    G_SystemInfo.DeviceName := SystemParameters.o_DeviceName;
    G_SystemInfo.HWVersion := SystemParameters.o_HardwareVersion;
    G_SystemInfo.SWVersion := SystemParameters.o_SoftwareVersion;
    G_SystemInfo.Identity.ProductCode := SystemParameters.o_ProductCode;    (* Type for control unit. *)
    G_SystemInfo.Identity.Revision := SystemParameters.o_RevisionNumber;      (* Revision for control unit *)
    G_SystemInfo.Identity.SerialNumber := SystemParameters.o_SerialNumber;  (* Serial number for control unit *)
    G_SystemInfo.Identity.VendorId := SystemParameters.o_VendorId;               (* Vendor id which is read from firmware *)
          
    G_SystemInfo.MACAddress := SystemParameters.o_MAC;
    G_SystemInfo.EthernetConfiguration :=  SystemParameters.i_Ethernet;
    G_SystemInfo.CAN1_Comms := SystemParameters.i_CAN1;
    G_SystemInfo.CAN2_Comms := SystemParameters.i_CAN2;
    G_SystemInfo.CAN3_Comms := SystemParameters.i_CAN3;
    G_SystemInfo.CAN4_Comms := SystemParameters.i_CAN4;
    
    (* Get 5050 fw error log pointer *)
    SystemErrorLog.init();
    G_SystemInfo.FWErrorLog :=  SystemErrorLog.o_ErrorLog;


    
END_IF
END_ACTION

ACTION Init_Events_Action:
(*###########################################################*)
(*This block is created implicit. Don't add own code to here.*)
(*###########################################################*)
;



G_InitEventsReady:=TRUE;
END_ACTION

ACTION Init_Exit_Action:
(*###########################################################*)
(*This block is created implicit. Don't add own code to here.*)
(*###########################################################*)
;


G_InitExitReady:=TRUE;
END_ACTION

ACTION Init_Flash_Action:
(*###########################################################*)
(*This block is created implicit. Don't add own code to here.*)
(*###########################################################*)

  	(* Get info for MRAM area used for programmer. *)
  	SYSTEM_SHM_MRAM_GET_IEC_AREA(ADR(G_ShmUserMRAM));
  	(* Check addresses and divide area between parameter system and are available for user *)
	IF ((G_ShmUserMRAM.endAddress > 0) AND (G_ShmUserMRAM.startAddress > 0))
		AND (G_ShmUserMRAM.endAddress > (G_ShmUserMRAM.startAddress + G_MRAM_AREA_SIZE_FOR_PAR_SYS + 100)) THEN
		(* Init file system for parameters *)
		(* Init ParameterHandler to use MRAM *)
        G_Common.ParHandler.Init(i_pParamArea:=G_ShmUserMRAM.startAddress,
            i_ParamAreaSize:=G_MRAM_AREA_SIZE_FOR_PAR_SYS ,
            i_Keyword:=G_PARAMHANDLERKEYWORD ,
            i_ParameterMaxDataSize:= G_PARAM_BLOCK_MAX_SIZE);
		(* Set user MRAM pointers, which tells area for freely used by programmer. *)
		G_MramStartAddressForUser := G_ShmUserMRAM.startAddress + G_MRAM_AREA_SIZE_FOR_PAR_SYS;
		G_MramEndAddressForUser := G_ShmUserMRAM.endAddress ;
	ELSE
		(* Error *)
		G_MramInitErrors := - 1;
	END_IF
	
	(* Init user MRAM structure*)
	IF (0 <> G_ShmUserMRAM.startAddress) AND (G_ShmUserMRAM.reservedSize >= (SIZEOF(UserMramStructure) + DWORD_TO_DINT(G_MRAM_AREA_SIZE_FOR_PAR_SYS))) THEN
		G_pUserMramStructure := G_MramStartAddressForUser;
		IF G_pUserMramStructure^.UserMRAMTag = 16#AA55AA55 THEN
			G_pUserMramStructure^.UserMRAMdataValid := TRUE;
			G_pUserMramStructure^.UserMRAMinitError := 0;
		ELSE
			G_pUserMramStructure^.UserMRAMdataValid := FALSE;
			G_pUserMramStructure^.UserMRAMTag := 16#AA55AA55;
			G_pUserMramStructure^.UserMRAMinitError := 2; 
		END_IF 
	END_IF
	
	
G_InitFlashReady:=TRUE;
END_ACTION

ACTION Init_IO_Action:
(*###########################################################*)
(*This block is created implicit. Don't add own code to here.*)
(*###########################################################*)
;
(*IO init:*)
(*IO_Init functions*)
		(* Force ref always ON *)
		REF_OUT_5V_Enable:=TRUE;
		REF_OUT_10V_Enable:=TRUE;

(*#########################################*)
(* INIT FOR AI Channel 1 X1.09*)

AI_SET_PU_u16_DrivetrainTemp_AI := FALSE;


    AI_SET_mA_u16_DrivetrainTemp_AI := FALSE;

    G_AIprotection_X1_09(i_Enable := TRUE, i_AiInmAMode:= FALSE);


(*#########################################*)
(* INIT FOR AI Channel 20 X1.10*)

    AI_SET_PU_u16_ChargePlugPresent_AI := FALSE;


    AI_SET_mA_u16_ChargePlugPresent_AI := FALSE;

    G_AIprotection_X1_10(i_Enable := TRUE, i_AiInmAMode:= FALSE);


(*##################################################################################*)
(* INIT FOR PULSE INPUT CHANNEL 22 Pin 1.11*)

PI_INIT_ERROR_q_BatteryInterlockIn_DI := IO_PULSEIN_SET_CONFIG(
	i_Mode:=IO_PULSEIN_MODE_DI,
	i_ChannelNbr:=22,
	i_ResetChnNbr:=0,
	i_ChannelPairNbr:=0,
	i_EdgeSelect:=0,
	i_EdgePolarity:=0,
	i_Filter:=0,
	i_GateTime:=100);
   IF NOT ( PI_INIT_ERROR_q_BatteryInterlockIn_DI = 0 ) THEN
         ERR_FLAG_IO_INIT := TRUE;
    END_IF

(*#########################################*)
(* INIT FOR PWFM CHANNEL 9 Pin 1.12*)

    PWFM_ERROR_INIT_q_BackupPump_DO :=  IO_PWFM_SET_CONFIG(
		i_PwfmMode:=IO_PWFM_MODE_DIGITAL_OUTPUT,
		i_PwfmChn:=9,
		i_OverCurrentLimit := 1000,
		i_SupplyVoltage:=0,
		i_CoilResistance:=0,
		i_CorrectionGain:=0,
		i_DiagnosticTimeDelay:=0);
   IF NOT ( PWFM_ERROR_INIT_q_BackupPump_DO = 0 ) THEN
         ERR_FLAG_IO_INIT := TRUE;
    END_IF
    DO_q_BackupPump_DO := FALSE;

(*#########################################*)
(* INIT FOR AI Channel 2 X1.20*)

    AI_SET_PU_u16_Heater1Temperature_AI := FALSE;


    AI_SET_mA_u16_Heater1Temperature_AI := FALSE;

    G_AIprotection_X1_20(i_Enable := TRUE, i_AiInmAMode:= FALSE);


(*#########################################*)
(* INIT FOR AI Channel 21 X1.21*)

    AI_SET_PU_u16_Heater2Temperature_AI := FALSE;


    AI_SET_mA_u16_Heater2Temperature_AI := FALSE;

    G_AIprotection_X1_21(i_Enable := TRUE, i_AiInmAMode:= FALSE);


(*#########################################*)
(* INIT FOR PWFM CHANNEL 21 Pin 1.22*)

    PWFM_ERROR_INIT_q_BatteryDischargeMain_DO := IO_PWFM_SET_CONFIG(
	i_PwfmMode:=IO_PWFM_MODE_DIGITAL_OUTPUT,
	i_PwfmChn:=21,
	i_OverCurrentLimit := 0,
	i_SupplyVoltage:=0,
	i_CoilResistance:=0,
	i_CorrectionGain:=0,
	i_DiagnosticTimeDelay:=0);
   IF NOT ( PWFM_ERROR_INIT_q_BatteryDischargeMain_DO = 0 ) THEN
         ERR_FLAG_IO_INIT := TRUE;
    END_IF
    DO_q_BatteryDischargeMain_DO := FALSE;

(*#########################################*)
(* INIT FOR PWFM CHANNEL 10 Pin 1.23*)

    PWFM_ERROR_INIT_q_AirPressureReliefValve_DO := IO_PWFM_SET_CONFIG(
	i_PwfmMode:=IO_PWFM_MODE_DIGITAL_OUTPUT,
	i_PwfmChn:=10,
	i_OverCurrentLimit := 1000,
	i_SupplyVoltage:=0,
	i_CoilResistance:=0,
	i_CorrectionGain:=0,
	i_DiagnosticTimeDelay:=0);
   IF NOT ( PWFM_ERROR_INIT_q_AirPressureReliefValve_DO = 0 ) THEN
         ERR_FLAG_IO_INIT := TRUE;
    END_IF
    DO_q_AirPressureReliefValve_DO := FALSE;

(*#########################################*)
(* INIT FOR PWFM CHANNEL 28 Pin 1.29*)

    PWFM_ERROR_INIT_q_Battery1ChargePrecharge_DO:= IO_PWFM_SET_CONFIG(
	i_PwfmMode:=IO_PWFM_MODE_DIGITAL_OUTPUT,
	i_PwfmChn:=28,
	i_OverCurrentLimit := 0,
	i_SupplyVoltage:=0,
	i_CoilResistance:=0,
	i_CorrectionGain:=0,
	i_DiagnosticTimeDelay:=0);
   IF NOT ( PWFM_ERROR_INIT_q_Battery1ChargePrecharge_DO = 0 ) THEN
         ERR_FLAG_IO_INIT := TRUE;
    END_IF
    DO_q_Battery1ChargePrecharge_DO := FALSE;

(*#########################################*)
(* INIT FOR PWFM CHANNEL 27 Pin 1.30*)

    PWFM_ERROR_INIT_q_Battery1ChargeMain_DO:= IO_PWFM_SET_CONFIG(
	i_PwfmMode:=IO_PWFM_MODE_DIGITAL_OUTPUT,
	i_PwfmChn:=27,
	i_OverCurrentLimit := 0,
	i_SupplyVoltage:=0,
	i_CoilResistance:=0,
	i_CorrectionGain:=0,
	i_DiagnosticTimeDelay:=0);
   IF NOT ( PWFM_ERROR_INIT_q_Battery1ChargeMain_DO = 0 ) THEN
         ERR_FLAG_IO_INIT := TRUE;
    END_IF
    DO_q_Battery1ChargeMain_DO := FALSE;

(*#########################################*)
(* INIT FOR PWFM CHANNEL 26 Pin 1.31*)

    PWFM_ERROR_INIT_q_Battery2ChargePrecharge_DO := IO_PWFM_SET_CONFIG(
	i_PwfmMode:=IO_PWFM_MODE_DIGITAL_OUTPUT,
	i_PwfmChn:=26,
	i_OverCurrentLimit := 0,
	i_SupplyVoltage:=0,
	i_CoilResistance:=0,
	i_CorrectionGain:=0,
	i_DiagnosticTimeDelay:=0);
   IF NOT ( PWFM_ERROR_INIT_q_Battery2ChargePrecharge_DO = 0 ) THEN
         ERR_FLAG_IO_INIT := TRUE;
    END_IF
    DO_q_Battery2ChargePrecharge_DO := FALSE;

(*#########################################*)
(* INIT FOR PWFM CHANNEL 25 Pin 1.32*)

    PWFM_ERROR_INIT_q_DrivetrainInverterTorqueless_DO := IO_PWFM_SET_CONFIG(
	i_PwfmMode:=IO_PWFM_MODE_DIGITAL_OUTPUT,
	i_PwfmChn:=25,
	i_OverCurrentLimit := 0,
	i_SupplyVoltage:=0,
	i_CoilResistance:=0,
	i_CorrectionGain:=0,
	i_DiagnosticTimeDelay:=0);
   IF NOT ( PWFM_ERROR_INIT_q_DrivetrainInverterTorqueless_DO = 0 ) THEN
         ERR_FLAG_IO_INIT := TRUE;
    END_IF
    DO_q_DrivetrainInverterTorqueless_DO := FALSE;

(*#########################################*)
(* INIT FOR PWFM CHANNEL 23 Pin 1.33*)

    PWFM_ERROR_INIT_q_BatteryDischargePrecharge_DO := IO_PWFM_SET_CONFIG(
	i_PwfmMode:=IO_PWFM_MODE_DIGITAL_OUTPUT,
	i_PwfmChn:=23,
	i_OverCurrentLimit := 0,
	i_SupplyVoltage:=0,
	i_CoilResistance:=0,
	i_CorrectionGain:=0,
	i_DiagnosticTimeDelay:=0);

   IF NOT ( PWFM_ERROR_INIT_q_BatteryDischargePrecharge_DO = 0 ) THEN
         ERR_FLAG_IO_INIT := TRUE;
    END_IF
	DO_q_BatteryDischargePrecharge_DO := FALSE;

(*#########################################*)
(* INIT FOR PWFM CHANNEL 24 Pin 1.34*)

    PWFM_ERROR_INIT_u32_DynamoFrequency_PWFM := IO_PWFM_SET_CONFIG(
	i_PwfmMode:=IO_PWFM_MODE_DIRECT_PWFM,
	i_PwfmChn:=24,
	i_OverCurrentLimit :=0,
	i_SupplyVoltage:=0,
	i_CoilResistance:=0,
	i_CorrectionGain:=0,
	i_DiagnosticTimeDelay:=0);
   IF NOT ( PWFM_ERROR_INIT_u32_DynamoFrequency_PWFM = 0 ) THEN
         ERR_FLAG_IO_INIT := TRUE;
    END_IF
    PWFM_FREQ_u32_DynamoFrequency_PWFM :=     200;
    PWFM_RATIO_u32_DynamoFrequency_PWFM := 0;

(*#########################################*)
(* INIT FOR PWFM CHANNEL 22 Pin 1.35*)

    PWFM_ERROR_INIT_q_Battery2ChargeMain_DO := IO_PWFM_SET_CONFIG(
	i_PwfmMode:=IO_PWFM_MODE_DIGITAL_OUTPUT,
	i_PwfmChn:=22,
	i_OverCurrentLimit := 0,
	i_SupplyVoltage:=0,
	i_CoilResistance:=0,
	i_CorrectionGain:=0,
	i_DiagnosticTimeDelay:=0);
   IF NOT ( PWFM_ERROR_INIT_q_Battery2ChargeMain_DO = 0 ) THEN
         ERR_FLAG_IO_INIT := TRUE;
    END_IF
    DO_q_Battery2ChargeMain_DO := FALSE;

(*##################################################################################*)
(* INIT FOR PULSE INPUT CHANNEL 1 Pin 2.6*)

PI_INIT_ERROR_q_Battery1ChargeRq_DI := IO_PULSEIN_SET_CONFIG(
	i_Mode:=IO_PULSEIN_MODE_1CH,
	i_ChannelNbr:=1,
	i_ResetChnNbr:=0,
	i_ChannelPairNbr:=0,
	i_EdgeSelect:=0,
	i_EdgePolarity:=0,
	i_Filter:=0,
	i_GateTime:=100);
   IF NOT ( PI_INIT_ERROR_q_Battery1ChargeRq_DI = 0 ) THEN
         ERR_FLAG_IO_INIT := TRUE;
    END_IF

(*##################################################################################*)
(* INIT FOR PULSE INPUT CHANNEL 2 Pin 2.7*)

    PI_INIT_ERROR_q_Battery1DiscahrgeRq_DI := IO_PULSEIN_SET_CONFIG(
	i_Mode:=IO_PULSEIN_MODE_1CH,
	i_ChannelNbr:=2,
	i_ResetChnNbr:=0,
	i_ChannelPairNbr:=0,
	i_EdgeSelect:=0,
	i_EdgePolarity:=0,
	i_Filter:=0,
	i_GateTime:=100);
    IF NOT ( PI_INIT_ERROR_q_Battery1DiscahrgeRq_DI = 0 ) THEN
         ERR_FLAG_IO_INIT := TRUE;
    END_IF

(*##################################################################################*)
(* INIT FOR PULSE INPUT CHANNEL 3 Pin 2.8*)

    PI_INIT_ERROR_q_Battery2ChargeRq_DI := IO_PULSEIN_SET_CONFIG(
	i_Mode:=IO_PULSEIN_MODE_1CH,
	i_ChannelNbr:=3,
	i_ResetChnNbr:=0,
	i_ChannelPairNbr:=0,
	i_EdgeSelect:=0,
	i_EdgePolarity:=0,
	i_Filter:=0,
	i_GateTime:=100);
   IF NOT ( PI_INIT_ERROR_q_Battery2ChargeRq_DI = 0 ) THEN
         ERR_FLAG_IO_INIT := TRUE;
    END_IF

(*##################################################################################*)
(* INIT FOR PULSE INPUT CHANNEL 4 Pin 2.9*)

    PI_INIT_ERROR_q_Batter2DischargeRq_DI := IO_PULSEIN_SET_CONFIG(
	i_Mode:=IO_PULSEIN_MODE_1CH,
	i_ChannelNbr:=4,
	i_ResetChnNbr:=0,
	i_ChannelPairNbr:=0,
	i_EdgeSelect:=0,
	i_EdgePolarity:=0,
	i_Filter:=0,
	i_GateTime:=100);
   IF NOT ( PI_INIT_ERROR_q_Batter2DischargeRq_DI = 0 ) THEN
         ERR_FLAG_IO_INIT := TRUE;
    END_IF

(*#########################################*)
(* INIT FOR PWFM CHANNEL 12 Pin 2.13*)

    PWFM_ERROR_INIT_q_ChargePlugLockPulse_DO := IO_PWFM_SET_CONFIG(
	i_PwfmMode:=IO_PWFM_MODE_DIGITAL_OUTPUT,
	i_PwfmChn:=12,
	i_OverCurrentLimit := 1000,
	i_SupplyVoltage:=0,
	i_CoilResistance:=0,
	i_CorrectionGain:=0,
	i_DiagnosticTimeDelay:=0);
    IF NOT ( PWFM_ERROR_INIT_q_ChargePlugLockPulse_DO = 0 ) THEN
         ERR_FLAG_IO_INIT := TRUE;
    END_IF
    DO_q_ChargePlugLockPulse_DO := FALSE;

(*#########################################*)
(* INIT FOR PWFM CHANNEL 11 Pin 2.14*)

    PWFM_ERROR_INIT_q_ChargePlugLockPosition_DO := IO_PWFM_SET_CONFIG(
	i_PwfmMode:=IO_PWFM_MODE_DIGITAL_OUTPUT,
	i_PwfmChn:=11,
	i_OverCurrentLimit := 1000,
	i_SupplyVoltage:=0,
	i_CoilResistance:=0,
	i_CorrectionGain:=0,
	i_DiagnosticTimeDelay:=0);
    IF NOT ( PWFM_ERROR_INIT_q_ChargePlugLockPosition_DO = 0 ) THEN
         ERR_FLAG_IO_INIT := TRUE;
    END_IF
    DO_q_ChargePlugLockPosition_DO := FALSE;

(*##################################################################################*)
(* INIT FOR PULSE INPUT CHANNEL 5 Pin 2.15*)

(*##################################################################################*)
(* INIT FOR PULSE INPUT CHANNEL 9 Pin 2.16*)

    PI_ERROR_q_ChargePlugLockStatus_DI := IO_PULSEIN_SET_CONFIG(
	i_Mode:=IO_PULSEIN_MODE_1CH,
	i_ChannelNbr:=9,
	i_ResetChnNbr:=0,
	i_ChannelPairNbr:=0,
	i_EdgeSelect:=0,
	i_EdgePolarity:=0,
	i_Filter:=0,
	i_GateTime:=100);
   IF NOT ( PI_ERROR_q_ChargePlugLockStatus_DI = 0 ) THEN
         ERR_FLAG_IO_INIT := TRUE;
    END_IF


(*##################################################################################*)
(* INIT FOR PULSE INPUT CHANNEL 10 Pin 2.17*)

(*##################################################################################*)
(* INIT FOR PULSE INPUT CHANNEL 6 Pin 2.18*)

(*##################################################################################*)
(* INIT FOR PULSE INPUT CHANNEL 11 Pin 2.19*)

(*##################################################################################*)
(* INIT FOR PULSE INPUT CHANNEL 12 Pin 2.20*)

(*#########################################*)
(* INIT FOR AI Channel 3 X2.23*)

    AI_SET_PU_u16_HeaterDiagnose_AI := FALSE;


    AI_SET_mA_u16_HeaterDiagnose_AI := FALSE;

    G_AIprotection_X2_23(i_Enable := TRUE, i_AiInmAMode:= FALSE);


(*#########################################*)
(* INIT FOR  SINKING DIGITAL OUTPUT 2.26*)

(*#########################################*)
(* INIT FOR  SINKING DIGITAL OUTPUT 2.27*)

(*#########################################*)
(* INIT FOR PWFM CHANNEL 14 Pin 2.28*)

    PWFM_ERROR_INIT_q_DrivetrainKL15D_DO := IO_PWFM_SET_CONFIG(
	i_PwfmMode:=IO_PWFM_MODE_DIGITAL_OUTPUT,
	i_PwfmChn:=14,
	i_OverCurrentLimit := 1000,
	i_SupplyVoltage:=0,
	i_CoilResistance:=0,
	i_CorrectionGain:=0,
	i_DiagnosticTimeDelay:=0);
    IF NOT ( PWFM_ERROR_INIT_q_DrivetrainKL15D_DO = 0 ) THEN
         ERR_FLAG_IO_INIT := TRUE;
    END_IF
    DO_q_DrivetrainKL15D_DO := FALSE;

(*#########################################*)
(* INIT FOR PWFM CHANNEL 13 Pin 2.29*)

    PWFM_ERROR_INIT_q_DrivetrainKL15C_DO := IO_PWFM_SET_CONFIG(
	i_PwfmMode:=IO_PWFM_MODE_DIGITAL_OUTPUT,
	i_PwfmChn:=13,
	i_OverCurrentLimit := 1000,
	i_SupplyVoltage:=0,
	i_CoilResistance:=0,
	i_CorrectionGain:=0,
	i_DiagnosticTimeDelay:=0);
    IF NOT ( PWFM_ERROR_INIT_q_DrivetrainKL15C_DO = 0 ) THEN
         ERR_FLAG_IO_INIT := TRUE;
    END_IF
    DO_q_DrivetrainKL15C_DO := FALSE;

(*#########################################*)
(* INIT FOR PWFM CHANNEL 16 Pin 2.30*)

    PWFM_ERROR_INIT_q_DrivetrainCoolingFan_DO := IO_PWFM_SET_CONFIG(
	i_PwfmMode:=IO_PWFM_MODE_DIGITAL_OUTPUT,
	i_PwfmChn:=16,
	i_OverCurrentLimit := 1000,
	i_SupplyVoltage:=0,
	i_CoilResistance:=0,
	i_CorrectionGain:=0,
	i_DiagnosticTimeDelay:=0);
    IF NOT ( PWFM_ERROR_INIT_q_DrivetrainCoolingFan_DO = 0 ) THEN
         ERR_FLAG_IO_INIT := TRUE;
    END_IF
    DO_q_DrivetrainCoolingFan_DO := FALSE;

(*#########################################*)
(* INIT FOR PWFM CHANNEL 15 Pin 2.31*)

    PWFM_ERROR_INIT_q_DrievtrainPowerSteering_DO := IO_PWFM_SET_CONFIG(
	i_PwfmMode:=IO_PWFM_MODE_DIGITAL_OUTPUT,
	i_PwfmChn:=15,
	i_OverCurrentLimit := 1000,
	i_SupplyVoltage:=0,
	i_CoilResistance:=0,
	i_CorrectionGain:=0,
	i_DiagnosticTimeDelay:=0);
    IF NOT ( PWFM_ERROR_INIT_q_DrievtrainPowerSteering_DO = 0 ) THEN
         ERR_FLAG_IO_INIT := TRUE;
    END_IF
    DO_q_DrievtrainPowerSteering_DO := FALSE;

(*#########################################*)
(* INIT FOR PWFM CHANNEL 18 Pin 2.32*)

    PWFM_ERROR_INIT_u32_HeaterControl_PWFM := IO_PWFM_SET_CONFIG(
	i_PwfmMode:=IO_PWFM_MODE_DIRECT_PWFM,
	i_PwfmChn:=18,
	i_OverCurrentLimit := 1000,
	i_SupplyVoltage:=0,
	i_CoilResistance:=0,
	i_CorrectionGain:=0,
	i_DiagnosticTimeDelay:=0);
    IF NOT ( PWFM_ERROR_INIT_u32_HeaterControl_PWFM = 0 ) THEN
         ERR_FLAG_IO_INIT := TRUE;
    END_IF
    PWFM_FREQ_u32_HeaterControl_PWFM :=     200;
    PWFM_RATIO_u32_HeaterControl_PWFM := 0;

(*#########################################*)
(* INIT FOR PWFM CHANNEL 17 Pin 2.33*)

    PWFM_ERROR_INIT_q_DrievtrainAirCompressor_DO := IO_PWFM_SET_CONFIG(
	i_PwfmMode:=IO_PWFM_MODE_DIGITAL_OUTPUT,
	i_PwfmChn:=17,
	i_OverCurrentLimit := 1000,
	i_SupplyVoltage:=0,
	i_CoilResistance:=0,
	i_CorrectionGain:=0,
	i_DiagnosticTimeDelay:=0);
    IF NOT ( PWFM_ERROR_INIT_q_DrievtrainAirCompressor_DO = 0 ) THEN
         ERR_FLAG_IO_INIT := TRUE;
    END_IF
    DO_q_DrievtrainAirCompressor_DO := FALSE;

(*#########################################*)
(* INIT FOR  SINKING DIGITAL OUTPUT 2.34*)

(*#########################################*)
(* INIT FOR  SINKING DIGITAL OUTPUT 2.35*)

DO_q_DynamoD_DO := FALSE;

(*##################################################################################*)
(* INIT FOR PULSE INPUT CHANNEL 17 Pin 3.5*)

    PI_INIT_ERROR_q_DirectionSwitch_ReverseCrawl_DI := IO_PULSEIN_SET_CONFIG(
	i_Mode:=IO_PULSEIN_MODE_DI,
	i_ChannelNbr:=17,
	i_ResetChnNbr:=0,
	i_ChannelPairNbr:=0,
	i_EdgeSelect:=0,
	i_EdgePolarity:=0,
	i_Filter:=0,
	i_GateTime:=100);
   IF NOT ( PI_INIT_ERROR_q_DirectionSwitch_ReverseCrawl_DI = 0 ) THEN
         ERR_FLAG_IO_INIT := TRUE;
    END_IF

(*##################################################################################*)
(* INIT FOR PULSE INPUT CHANNEL 18 Pin 3.6*)

    PI_INIT_ERROR_q_DirectionSwitch_Drive_DI := IO_PULSEIN_SET_CONFIG(
	i_Mode:=IO_PULSEIN_MODE_DI,
	i_ChannelNbr:=18,
	i_ResetChnNbr:=0,
	i_ChannelPairNbr:=0,
	i_EdgeSelect:=0,
	i_EdgePolarity:=0,
	i_Filter:=0,
	i_GateTime:=100);
   IF NOT ( PI_INIT_ERROR_q_DirectionSwitch_Drive_DI = 0 ) THEN
         ERR_FLAG_IO_INIT := TRUE;
    END_IF

(*##################################################################################*)
(* INIT FOR PULSE INPUT CHANNEL 7 Pin 3.7*)

    PI_ERROR_q_IlluminiationStatsus_DI := IO_PULSEIN_SET_CONFIG(
	i_Mode:=IO_PULSEIN_MODE_1CH,
	i_ChannelNbr:=7,
	i_ResetChnNbr:=0,
	i_ChannelPairNbr:=0,
	i_EdgeSelect:=0,
	i_EdgePolarity:=0,
	i_Filter:=0,
	i_GateTime:=100);
    IF NOT ( PI_ERROR_q_IlluminiationStatsus_DI = 0 ) THEN
         ERR_FLAG_IO_INIT := TRUE;
    END_IF

(*##################################################################################*)
(* INIT FOR PULSE INPUT CHANNEL 13 Pin 3.8*)

    PI_INIT_ERROR_q_DirectionSwitch_Reverse_DI := IO_PULSEIN_SET_CONFIG(
	i_Mode:=IO_PULSEIN_MODE_DI,
	i_ChannelNbr:=13,
	i_ResetChnNbr:=0,
	i_ChannelPairNbr:=0,
	i_EdgeSelect:=0,
	i_EdgePolarity:=0,
	i_Filter:=0,
	i_GateTime:=100);
    IF NOT ( PI_INIT_ERROR_q_DirectionSwitch_Reverse_DI = 0 ) THEN
         ERR_FLAG_IO_INIT := TRUE;
    END_IF

(*##################################################################################*)
(* INIT FOR PULSE INPUT CHANNEL 14 Pin 3.9*)

    PI_INIT_ERROR_q_DirectionSwitch_DriveCrawl_DI := IO_PULSEIN_SET_CONFIG(
	i_Mode:=IO_PULSEIN_MODE_DI,
	i_ChannelNbr:=14,
	i_ResetChnNbr:=0,
	i_ChannelPairNbr:=0,
	i_EdgeSelect:=0,
	i_EdgePolarity:=0,
	i_Filter:=0,
	i_GateTime:=100);
    IF NOT ( PI_INIT_ERROR_q_DirectionSwitch_DriveCrawl_DI = 0 ) THEN
         ERR_FLAG_IO_INIT := TRUE;
    END_IF

(*##################################################################################*)
(* INIT FOR PULSE INPUT CHANNEL 8 Pin 3.10*)

(*##################################################################################*)
(* INIT FOR PULSE INPUT CHANNEL 15 Pin 3.11*)

    PI_INIT_ERROR_q_DirectionSwitch_Neutral_DI := IO_PULSEIN_SET_CONFIG(
	i_Mode:=IO_PULSEIN_MODE_DI,
	i_ChannelNbr:=15,
	i_ResetChnNbr:=0,
	i_ChannelPairNbr:=0,
	i_EdgeSelect:=0,
	i_EdgePolarity:=0,
	i_Filter:=0,
	i_GateTime:=100);
    IF NOT ( PI_INIT_ERROR_q_DirectionSwitch_Neutral_DI = 0 ) THEN
         ERR_FLAG_IO_INIT := TRUE;
    END_IF

(*##################################################################################*)
(* INIT FOR PULSE INPUT CHANNEL 16 Pin 3.12*)

    PI_INIT_ERROR_q_DoorOpen_DI := IO_PULSEIN_SET_CONFIG(
	i_Mode:=IO_PULSEIN_MODE_DI,
	i_ChannelNbr:=16,
	i_ResetChnNbr:=0,
	i_ChannelPairNbr:=0,
	i_EdgeSelect:=0,
	i_EdgePolarity:=0,
	i_Filter:=0,
	i_GateTime:=100);
    IF NOT ( PI_INIT_ERROR_q_DoorOpen_DI = 0 ) THEN
         ERR_FLAG_IO_INIT := TRUE;
    END_IF

(*#########################################*)
(* INIT FOR AI Channel 22 X3.14*)

    AI_SET_PU_u16_HeaterDiagnose2_AI := FALSE;


    AI_SET_mA_u16_HeaterDiagnose2_AI := FALSE;

    G_AIprotection_X3_14(i_Enable := TRUE, i_AiInmAMode:= FALSE);


(*#########################################*)
(* INIT FOR AI Channel 4 X3.15*)

    AI_SET_PU_u16_VehicleThrottlePedal1_AI := FALSE;


    AI_SET_mA_u16_VehicleThrottlePedal1_AI := FALSE;

    G_AIprotection_X3_15(i_Enable := TRUE, i_AiInmAMode:= FALSE);


(*#########################################*)
(* INIT FOR AI Channel 4 X3.15*)

    AI_SET_PU_u16_VehicleThrottlePedal2_AI := FALSE;


    AI_SET_mA_u16_VehicleThrottlePedal2_AI := FALSE;

    G_AIprotection_X3_16(i_Enable := TRUE, i_AiInmAMode:= FALSE);


(*##################################################################################*)
(* INIT FOR PULSE INPUT CHANNEL 19 Pin 3.21*)

(*##################################################################################*)
(* INIT FOR PULSE INPUT CHANNEL 20 Pin 3.22*)

    PI_INIT_ERROR_q_VehicleKL15_DI := IO_PULSEIN_SET_CONFIG(
	i_Mode:=IO_PULSEIN_MODE_DI,
	i_ChannelNbr:=20,
	i_ResetChnNbr:=0,
	i_ChannelPairNbr:=0,
	i_EdgeSelect:=0,
	i_EdgePolarity:=0,
	i_Filter:=0,
	i_GateTime:=100);
    IF NOT ( PI_INIT_ERROR_q_VehicleKL15_DI = 0 ) THEN
         ERR_FLAG_IO_INIT := TRUE;
    END_IF

(*##################################################################################*)
(* INIT FOR PULSE INPUT CHANNEL 21 Pin 3.23*)

    PI_INIT_ERROR_q_VehicleKL51_DI := IO_PULSEIN_SET_CONFIG(
	i_Mode:=IO_PULSEIN_MODE_DI,
	i_ChannelNbr:=21,
	i_ResetChnNbr:=0,
	i_ChannelPairNbr:=0,
	i_EdgeSelect:=0,
	i_EdgePolarity:=0,
	i_Filter:=0,
	i_GateTime:=100);
    IF NOT ( PI_INIT_ERROR_q_VehicleKL51_DI = 0 ) THEN
         ERR_FLAG_IO_INIT := TRUE;
    END_IF

(*#########################################*)
(* INIT FOR PWFM CHANNEL 20 Pin 3.26*)

    PWFM_ERROR_INIT_q_ChargersWakeup_DO := IO_PWFM_SET_CONFIG(
	i_PwfmMode:=IO_PWFM_MODE_DIGITAL_OUTPUT,
	i_PwfmChn:=20,
	i_OverCurrentLimit := 1000,
	i_SupplyVoltage:=0,
	i_CoilResistance:=0,
	i_CorrectionGain:=0,
	i_DiagnosticTimeDelay:=0);
    IF NOT ( PWFM_ERROR_INIT_q_ChargersWakeup_DO = 0 ) THEN
         ERR_FLAG_IO_INIT := TRUE;
    END_IF
    DO_q_ChargersWakeup_DO := FALSE;

(*#########################################*)
(* INIT FOR PWFM CHANNEL 19 Pin 3.27*)

    PWFM_ERROR_INIT_q_DashboardDCDCStatus_DO := IO_PWFM_SET_CONFIG(
	i_PwfmMode:=IO_PWFM_MODE_DIGITAL_OUTPUT,
	i_PwfmChn:=19,
	i_OverCurrentLimit := 1000,
	i_SupplyVoltage:=0,
	i_CoilResistance:=0,
	i_CorrectionGain:=0,
	i_DiagnosticTimeDelay:=0);
    IF NOT ( PWFM_ERROR_INIT_q_DashboardDCDCStatus_DO = 0 ) THEN
         ERR_FLAG_IO_INIT := TRUE;
    END_IF
    DO_q_DashboardDCDCStatus_DO := FALSE;

(*#########################################*)
(* INIT FOR PWFM CHANNEL 2 Pin 3.28*)

    PWFM_ERROR_INIT_q_HeaterIn_DI := IO_PWFM_SET_CONFIG(
	i_PwfmMode:=IO_PWFM_MODE_DISABLED,
	i_PwfmChn:=2,
	i_OverCurrentLimit := 100,
	i_SupplyVoltage:=0,
	i_CoilResistance:=0,
	i_CorrectionGain:=0,
	i_DiagnosticTimeDelay:=0);
    IF NOT ( PWFM_ERROR_INIT_q_HeaterIn_DI = 0 ) THEN
         ERR_FLAG_IO_INIT := TRUE;
    END_IF

(*#########################################*)
(* INIT FOR PWFM CHANNEL 1 Pin 3.29 *)

    PWFM_ERROR_INIT_q_HeaterOut_DI := IO_PWFM_SET_CONFIG(
	i_PwfmMode:=IO_PWFM_MODE_DIGITAL_OUTPUT,
	i_PwfmChn:=1,
	i_OverCurrentLimit := 1000,
	i_SupplyVoltage:=0,
	i_CoilResistance:=0,
	i_CorrectionGain:=0,
	i_DiagnosticTimeDelay:=100);
    IF NOT ( PWFM_ERROR_INIT_q_HeaterOut_DI = 0 ) THEN
         ERR_FLAG_IO_INIT := TRUE;
    END_IF
    DO_q_HeaterOut_DI := FALSE;

(*#########################################*)
(* INIT FOR PWFM CHANNEL 4 Pin 3.30*)

    PWFM_ERROR_INIT_q_DrivetrainInverterRf1_DO := IO_PWFM_SET_CONFIG(
	i_PwfmMode:=IO_PWFM_MODE_DIGITAL_OUTPUT,
	i_PwfmChn:=4,
	i_OverCurrentLimit := 1000,
	i_SupplyVoltage:=0,
	i_CoilResistance:=0,
	i_CorrectionGain:=0,
	i_DiagnosticTimeDelay:=0);
    IF NOT ( PWFM_ERROR_INIT_q_DrivetrainInverterRf1_DO = 0 ) THEN
         ERR_FLAG_IO_INIT := TRUE;
    END_IF
    DO_q_DrivetrainInverterRf1_DO := FALSE;

(*#########################################*)
(* INIT FOR PWFM CHANNEL 3 Pin 3.31*)

    PWFM_ERROR_INIT_q_DrivetrainInverterRf2_DO := IO_PWFM_SET_CONFIG(
	i_PwfmMode:=IO_PWFM_MODE_DIGITAL_OUTPUT,
	i_PwfmChn:=3,
	i_OverCurrentLimit := 1000,
	i_SupplyVoltage:=0,
	i_CoilResistance:=0,
	i_CorrectionGain:=0,
	i_DiagnosticTimeDelay:=0);
    IF NOT ( PWFM_ERROR_INIT_q_DrivetrainInverterRf2_DO = 0 ) THEN
         ERR_FLAG_IO_INIT := TRUE;
    END_IF
    DO_q_DrivetrainInverterRf2_DO := FALSE;

(*#########################################*)
(* INIT FOR PWFM CHANNEL 6 Pin 3.32*)

    PWFM_ERROR_INIT_q_DrivetrainDCDCInhibit_DO := IO_PWFM_SET_CONFIG(
	i_PwfmMode:=IO_PWFM_MODE_DIGITAL_OUTPUT,
	i_PwfmChn:=6,
	i_OverCurrentLimit := 1000,
	i_SupplyVoltage:=0,
	i_CoilResistance:=0,
	i_CorrectionGain:=0,
	i_DiagnosticTimeDelay:=0);
    IF NOT ( PWFM_ERROR_INIT_q_DrivetrainDCDCInhibit_DO = 0 ) THEN
         ERR_FLAG_IO_INIT := TRUE;
    END_IF
    DO_q_DrivetrainDCDCInhibit_DO := FALSE;

(*#########################################*)
(* INIT FOR PWFM CHANNEL 5 Pin 3.33*)

    PWFM_ERROR_INIT_q_ChargePlugLED_Green_DO := IO_PWFM_SET_CONFIG(
	i_PwfmMode:=IO_PWFM_MODE_DIGITAL_OUTPUT,
	i_PwfmChn:=5,
	i_OverCurrentLimit := 1000,
	i_SupplyVoltage:=0,
	i_CoilResistance:=0,
	i_CorrectionGain:=0,
	i_DiagnosticTimeDelay:=0);
    IF NOT ( PWFM_ERROR_INIT_q_ChargePlugLED_Green_DO = 0 ) THEN
         ERR_FLAG_IO_INIT := TRUE;
    END_IF
    DO_q_ChargePlugLED_Green_DO := FALSE;

(*#########################################*)
(* INIT FOR PWFM CHANNEL 8 Pin 3.34*)

    PWFM_ERROR_INIT_q_ChargePlugLED_Blue_DO := IO_PWFM_SET_CONFIG(
	i_PwfmMode:=IO_PWFM_MODE_DIGITAL_OUTPUT,
	i_PwfmChn:=8,
	i_OverCurrentLimit := 1000,
	i_SupplyVoltage:=0,
	i_CoilResistance:=0,
	i_CorrectionGain:=0,
	i_DiagnosticTimeDelay:=0);
    IF NOT ( PWFM_ERROR_INIT_q_ChargePlugLED_Blue_DO = 0 ) THEN
         ERR_FLAG_IO_INIT := TRUE;
    END_IF
    DO_q_ChargePlugLED_Blue_DO := FALSE;

(*#########################################*)
(* INIT FOR PWFM CHANNEL 7 Pin 3.35*)

    PWFM_ERROR_INIT_q_ChargePlugLED_Red_DO := IO_PWFM_SET_CONFIG(
	i_PwfmMode:=IO_PWFM_MODE_DIGITAL_OUTPUT,
	i_PwfmChn:=7,
	i_OverCurrentLimit := 1000,
	i_SupplyVoltage:=0,
	i_CoilResistance:=0,
	i_CorrectionGain:=0,
	i_DiagnosticTimeDelay:=0);
    IF NOT ( PWFM_ERROR_INIT_q_ChargePlugLED_Red_DO = 0 ) THEN
         ERR_FLAG_IO_INIT := TRUE;
    END_IF
    DO_q_ChargePlugLED_Red_DO := FALSE;

(*#########################################*)

    (* SET PULL UP CONFIGURATION *)

    PWFM_SET_PU_1_22_and_1_35 := FALSE;
    PWFM_SET_PU_1_33_and_1_34 := FALSE;
    PWFM_SET_PU_1_31_and_1_32 := FALSE;
    PWFM_SET_PU_1_29_and_1_30 := FALSE;
    PI_SET_PU_2_06_and_2_07 := FALSE;
    PI_SET_PU_2_08_and_2_09 := FALSE;
    PI_SET_PU_3_05_and_3_06 := FALSE;
    PI_SET_PU_3_08_and_3_09 := FALSE;
    PI_SET_PU_3_11_and_3_12 := FALSE;
    PI_SET_PU_3_21_and_3_22 := FALSE;
    PI_SET_PU_1_11_and_3_23 := FALSE;
    PI_SET_PU_2_16_and_2_17 := FALSE;
    PI_SET_PU_2_19_and_2_20 := FALSE;


(*#########################################*)
    (* SET Range configuration *)
    PI_SET_RANGE_2_06_and_2_07 := FALSE;
    PI_SET_RANGE_2_08_and_2_09 := FALSE;


(*IO-init OK?*)
G_InitIOReady:=TRUE;
END_ACTION

ACTION Init_Protocols_Can1_Action:
(*###########################################################*)
(*This block is created implicit. Don't add own code to here.*)
(*###########################################################*)
;
CASE G_InitProtocolsCan1State OF

InitCanProtocolStates.INIT_CANOPEN_PROTOCOLS:
(*CAN1 INIT*)

G_CANopen_CAN1.Device.itfCanChannel:=G_CAN1_Channel; (*Connect device to can channel*)
G_CANopen_CAN1.Device.NodeID := BYTE#1;
G_CANopen_CAN1.NMT.NmtState:=EPEC_CANopen.NMTState.BootUp; (* Set NMT status to BOOTUP *)

(*Initialize OD's data structures*)
G_CANopen_CAN1.OD.EntryCount:=SIZEOF(G_CANopen_CAN1.ODEntrys)/SIZEOF(G_CANopen_CAN1.ODEntrys[1]); (*Max entries of given OD(CANopenDeviceODEntrys array)*)
G_CANopen_CAN1.OD.InOrder:=FALSE; (*OD isn't in order*)
G_CANopen_CAN1.OD.NextFree:=0; (*OD does not have any entries yet*)
G_CANopen_CAN1.OD.pODEntry:=ADR(G_CANopen_CAN1.ODEntrys); (*Pointer to OD array*)

(*Define NMT protocol*)
G_CANopen_CAN1.Protocols[1].Protocol:=EPEC_CANopen.ProtocolType.NMT;
G_CANopen_CAN1.Protocols[1].pData:=ADR(G_CANopen_CAN1.NMT);
G_CANopen_CAN1.Protocols[1].itfProtocol:=G_CANopen_CAN1.NMT_Handler;
G_CANopen_CAN1.Protocols[1].pError:=ADR(G_CANopen_CAN1_VAR.NMT_Error);
G_CANopen_CAN1_VAR.ProtocolAdded[1] := CANopenDeviceAddProtocol( (* Add to protocol stack *)
	i_pDevice:=ADR(G_CANopen_CAN1.Device),
	i_pProtocol:=ADR(G_CANopen_CAN1.Protocols[1]),
);

(*Initialize NMT protocol*)
IF G_CANopen_CAN1_VAR.ProtocolAdded[1] THEN
	G_CANopen_CAN1.NMT_Handler.Init(
		i_pDevice := ADR(G_CANopen_CAN1.Device),
		i_ThisIsMaster := FALSE,
		i_StartInterval :=  1000,
		i_pMonitoredNodes := 0,
		i_NumberOfNodes := 0,
		i_SimultaneousSlaveConfiguration := FALSE,
		o_Error => G_CANopen_CAN1_VAR.NMT_Error
	);
ELSE
	G_CANopen_CAN1_VAR.NMT_Error := EPEC_CANopen.Errors.ProtocolDataMissing;
END_IF

(*Define OD protocol*)
G_CANopen_CAN1.Protocols[2].Protocol:=EPEC_CANopen.ProtocolType.OD;
G_CANopen_CAN1.Protocols[2].pData:=ADR(G_CANopen_CAN1.OD);
G_CANopen_CAN1.Protocols[2].pError:=ADR(G_CANopen_CAN1_VAR.OD_Error);
G_CANopen_CAN1_VAR.ProtocolAdded[2] := CANopenDeviceAddProtocol( (* Add to protocol stack *)
	i_pDevice:=ADR(G_CANopen_CAN1.Device),
	i_pProtocol:=ADR(G_CANopen_CAN1.Protocols[2]),
);
IF NOT G_CANopen_CAN1_VAR.ProtocolAdded[2] THEN
	G_CANopen_CAN1_VAR.OD_Error := EPEC_CANopen.Errors.ProtocolDataMissing;
END_IF

(*Define HB protocol
- Uses NMT and OD protocol data, thus need to be defined after them.
*)
G_CANopen_CAN1.HB.HeartBeat.PT := T#200MS; (* HB producer time *)

G_CANopen_CAN1.Protocols[3].Protocol:=EPEC_CANopen.ProtocolType.HB;
G_CANopen_CAN1.Protocols[3].pData:=ADR(G_CANopen_CAN1.HB);
G_CANopen_CAN1.Protocols[3].itfProtocol:=G_CANopen_CAN1.HB_Handler;
G_CANopen_CAN1.Protocols[3].pError:=ADR(G_CANopen_CAN1_VAR.HB_Error);
G_CANopen_CAN1_VAR.ProtocolAdded[3] := CANopenDeviceAddProtocol( (* Add to protocol stack *)
	i_pDevice:=ADR(G_CANopen_CAN1.Device),
	i_pProtocol:=ADR(G_CANopen_CAN1.Protocols[3]),
);

(* Initialize HB protocol *)
IF G_CANopen_CAN1_VAR.ProtocolAdded[3] THEN
	G_CANopen_CAN1.HB_Handler.Init(
		i_pDevice := ADR(G_CANopen_CAN1.Device),
		o_Error => G_CANopen_CAN1_VAR.HB_Error
	);

	(* Add monitored nodes *)
ELSE
	G_CANopen_CAN1_VAR.HB_Error := EPEC_CANopen.Errors.ProtocolDataMissing;
END_IF

(*Define SSDO protocol*)
G_CANopen_CAN1.Protocols[4].Protocol:=EPEC_CANopen.ProtocolType.SSDO;
G_CANopen_CAN1.Protocols[4].pData:=ADR(G_CANopen_CAN1.SSDO);
G_CANopen_CAN1.Protocols[4].itfProtocol:=G_CANopen_CAN1.SSDO_Handler;
G_CANopen_CAN1.Protocols[4].pError:=ADR(G_CANopen_CAN1_VAR.SSDO_Error);
G_CANopen_CAN1_VAR.ProtocolAdded[4] := CANopenDeviceAddProtocol( (* Add to protocol stack *)
	i_pDevice:=ADR(G_CANopen_CAN1.Device),
	i_pProtocol:=ADR(G_CANopen_CAN1.Protocols[4])
);
IF G_CANopen_CAN1_VAR.ProtocolAdded[4] THEN
	G_CANopen_CAN1.SSDO_Handler.Init(
		i_pDevice := ADR(G_CANopen_CAN1.Device),
		o_Error => G_CANopen_CAN1_VAR.SSDO_Error
	);
ELSE
	G_CANopen_CAN1_VAR.SSDO_Error := EPEC_CANopen.Errors.ProtocolDataMissing;
END_IF

(*Define GFC protocol*)
G_CANopen_CAN1.Protocols[5].Protocol:=EPEC_CANopen.ProtocolType.GFC;
G_CANopen_CAN1.Protocols[5].pData:=ADR(G_CANopen_CAN1.GFC);
G_CANopen_CAN1.Protocols[5].itfProtocol:=G_CANopen_CAN1.GFC_Handler;
G_CANopen_CAN1.Protocols[5].pError:=ADR(G_CANopen_CAN1_VAR.GFC_Error);
G_CANopen_CAN1_VAR.ProtocolAdded[5] := CANopenDeviceAddProtocol(  (* Add to protocol stack *)
	i_pDevice:=ADR(G_CANopen_CAN1.Device),
	i_pProtocol:=ADR(G_CANopen_CAN1.Protocols[5])
);
IF G_CANopen_CAN1_VAR.ProtocolAdded[5] THEN
	G_CANopen_CAN1.GFC_Handler.Init(
		i_pDevice := ADR(G_CANopen_CAN1.Device),
		i_pStatus:=ADR(G_CANopen_CAN1_VAR.GFC_Status),
		o_Error => G_CANopen_CAN1_VAR.GFC_Error
	);
ELSE
	G_CANopen_CAN1_VAR.GFC_Error := EPEC_CANopen.Errors.ProtocolDataMissing;
END_IF

(* Init CSDO instance array for bus *)
EPEC_CANopen.CANopenSDOManager.Init(
	i_pDevice:=ADR(G_CANopen_CAN1.Device),
	i_NodeId:=G_CANopen_CAN1.Device.NodeID,
	i_pCsdoArrayStart:=ADR(G_CANopen_CAN1.CSDOS),
	i_CsdoArraySize:=127,
	o_Error=>G_CANopen_CAN1_VAR.CSDO_Error
);





G_InitProtocolsCan1State := InitCanProtocolStates.INIT_CANOPEN_OD;

InitCanProtocolStates.INIT_CANOPEN_OD:

(*16#0001..16#0009 Default types *)
G_CANopen_CAN1_VAR.OD_Error := EPEC_CANopen.CANopenODAddDefautTypes(
	i_pOD:= ADR(G_CANopen_CAN1.OD)
);

(* 16#1000 Information about the device type *)
IF G_CANopen_CAN1_VAR.OD_Error = EPEC_CANopen.Errors.NoError THEN
	G_CANopen_CAN1_VAR.OD_Error := CANopenODAddLine(
		i_pOD := ADR(G_CANopen_CAN1.OD),(*Address of Object dictionary where index will be added*)
		i_Index := G_CANOPEN_ODINDEX_DEVICE_TYPE,
		i_ObjectCode := EPEC_CANopen.ObjectCode.OD_VAR,(*Type of index*)
		i_NumOfSubids := USINT#0,(*Number of subindexes*)
		i_TypeSpec := EPEC_CANopen.DataType.Deftype_UNSIGNED32,(*Index datatype, either user defined or standard CiA 301*)
		i_ObjectAccess := G_CANOPEN_OD_ACCESS_NOWRITE OR G_CANOPEN_OD_ACCESS_SUB0NOWRITE,
		i_Sub0data := USINT#0,(*Value of subindex0 in array or (def)struct*)
		i_pIndexData := ADR(G_CAN1_VAR.DeviceType_Device1),
		i_itfSDOHandler := DWORD#0
	);
END_IF

(* 16#1001 Error information *)
IF G_CANopen_CAN1_VAR.OD_Error = EPEC_CANopen.Errors.NoError THEN
	G_CANopen_CAN1_VAR.OD_Error := CANopenODAddLine(
		i_pOD := ADR(G_CANopen_CAN1.OD),(*Address of Object dictionary where index will be added*)
		i_Index := G_CANOPEN_ODINDEX_ERROR_REGISTER,
		i_ObjectCode := EPEC_CANopen.ObjectCode.OD_VAR,(*Type of index*)
		i_NumOfSubids := USINT#0,(*Number of subindexes*)
		i_TypeSpec := EPEC_CANopen.DataType.Deftype_UNSIGNED8,(*Index datatype, either user defined or standard CiA 301*)
		i_ObjectAccess := G_CANOPEN_OD_ACCESS_NOWRITE OR G_CANOPEN_OD_ACCESS_SUB0NOWRITE,
		i_Sub0data := USINT#0,(*Value of subindex0 in array or (def)struct*)
		i_pIndexData := ADR(G_CAN1_VAR.ErrorReg_Device1),
		i_itfSDOHandler := DWORD#0
	);
END_IF

(* 16#1008 Manufacturer device name *)
IF G_CANopen_CAN1_VAR.OD_Error = EPEC_CANopen.Errors.NoError THEN
	G_CANopen_CAN1_VAR.OD_Error := CANopenODAddLine(
		i_pOD := ADR(G_CANopen_CAN1.OD),(*Address of Object dictionary where index will be added*)
		i_Index := G_CANOPEN_ODINDEX_MF_DEVICE_NAME,
		i_ObjectCode := EPEC_CANopen.ObjectCode.OD_VAR,(*Type of index*)
		i_NumOfSubids := USINT#0,(*Number of subindexes*)
		i_TypeSpec := EPEC_CANopen.DataType.Deftype_STRING,(*Index datatype, either user defined or standard CiA 301*)
		i_ObjectAccess := G_CANOPEN_OD_ACCESS_NOWRITE OR G_CANOPEN_OD_ACCESS_SUB0NOWRITE,
		i_Sub0data := USINT#0,(*Value of subindex0 in array or (def)struct*)
		i_pIndexData := ADR(G_SystemInfo.DeviceName),
		i_itfSDOHandler := DWORD#0
	);
END_IF

(* 16#100A Manufacturer software version *)
IF G_CANopen_CAN1_VAR.OD_Error = EPEC_CANopen.Errors.NoError THEN
	G_CANopen_CAN1_VAR.OD_Error := CANopenODAddLine(
		i_pOD := ADR(G_CANopen_CAN1.OD),(*Address of Object dictionary where index will be added*)
		i_Index := G_CANOPEN_ODINDEX_MF_SW_VERSION,
		i_ObjectCode := EPEC_CANopen.ObjectCode.OD_VAR,(*Type of index*)
		i_NumOfSubids := USINT#0,(*Number of subindexes*)
		i_TypeSpec := EPEC_CANopen.DataType.Deftype_STRING,(*Index datatype, either user defined or standard CiA 301*)
		i_ObjectAccess := G_CANOPEN_OD_ACCESS_NOWRITE OR G_CANOPEN_OD_ACCESS_SUB0NOWRITE,
		i_Sub0data := USINT#0,(*Value of subindex0 in array or (def)struct*)
		i_pIndexData := ADR(G_SystemInfo.SWVersion),
		i_itfSDOHandler := DWORD#0
	);
END_IF

(* 16#1018   Vendor ID *)
IF G_CANopen_CAN1_VAR.OD_Error = EPEC_CANopen.Errors.NoError THEN
	G_CANopen_CAN1_VAR.OD_Error := CANopenODAddLine(
		i_pOD := ADR(G_CANopen_CAN1.OD),(*Address of Object dictionary where index will be added*)
		i_index := G_CANOPEN_ODINDEX_IDENTITY_OBJECT,
		i_ObjectCode := EPEC_CANopen.ObjectCode.OD_ARRAY, (*Type of index*)
		i_NumOfSubids := USINT#4,(*Number of subindexes*)
		i_TypeSpec := EPEC_CANopen.DataType.Deftype_UNSIGNED32,(*Index of 16-bit deftype*)
		i_ObjectAccess := G_CANOPEN_OD_ACCESS_NOWRITE OR G_CANOPEN_OD_ACCESS_SUB0NOWRITE,
		i_sub0data := USINT#4,(*Value of subindex0 in array or (def)struct*)
		i_pIndexData := ADR(G_SystemInfo.Identity),
		i_itfSDOHandler := DWORD#0
	);
END_IF
(* 16#2030   CodesysVersion *)
IF G_CANopen_CAN1_VAR.OD_Error = EPEC_CANopen.Errors.NoError THEN
	G_CANopen_CAN1_VAR.OD_Error := CANopenODAddLine(
		i_pOD := ADR(G_CANopen_CAN1.OD),(*Address of Object dictionary where index will be added*)
		i_index := 16#2030,
		i_ObjectCode := EPEC_CANopen.ObjectCode.OD_ARRAY, (*Type of index*)
		i_NumOfSubids := USINT#1,(*Number of subindexes*)
		i_TypeSpec := EPEC_CANopen.DataType.Deftype_UNSIGNED32,(*Index of 16-bit deftype*)
		i_ObjectAccess := G_CANOPEN_OD_ACCESS_READWRITE OR G_CANOPEN_OD_ACCESS_SUB0NOWRITE,
		i_sub0data := USINT#1,(*Value of subindex0 in array or (def)struct*)
		i_pIndexData := ADR(G_SystemInfo.ToolsVersionInfo),
		i_itfSDOHandler := DWORD#0
	);
END_IF

(* 16#2128 PDO Dummy Variable Index *)
IF G_CANopen_CAN1_VAR.OD_Error = EPEC_CANopen.Errors.NoError THEN
	G_CANopen_CAN1_VAR.OD_Error := CANopenODAddLine(
		i_pOD := ADR(G_CANopen_CAN1.OD),(*Address of Object dictionary where index will be added*)
		i_Index := 16#2128,
		i_ObjectCode := EPEC_CANopen.ObjectCode.OD_VAR,(*Type of index*)
		i_NumOfSubids := USINT#0,(*Number of subindexes*)
		i_TypeSpec := EPEC_CANopen.DataType.Deftype_UNSIGNED8,(*Index datatype, either user defined or standard CiA 301*)
		i_ObjectAccess := G_CANOPEN_OD_ACCESS_READWRITE,
		i_Sub0data := USINT#0,(*Value of subindex0 in array or (def)struct*)
		i_pIndexData := ADR(G_CAN1_VAR.CAN1_TPDO_DUMMY),
		i_itfSDOHandler := DWORD#0
	);
END_IF

(* 16#2129 PDO Dummy Variable Index *)
IF G_CANopen_CAN1_VAR.OD_Error = EPEC_CANopen.Errors.NoError THEN
	G_CANopen_CAN1_VAR.OD_Error := CANopenODAddLine(
		i_pOD := ADR(G_CANopen_CAN1.OD),(*Address of Object dictionary where index will be added*)
		i_Index := 16#2129,
		i_ObjectCode := EPEC_CANopen.ObjectCode.OD_VAR,(*Type of index*)
		i_NumOfSubids := USINT#0,(*Number of subindexes*)
		i_TypeSpec := EPEC_CANopen.DataType.Deftype_UNSIGNED8,(*Index datatype, either user defined or standard CiA 301*)
		i_ObjectAccess := G_CANOPEN_OD_ACCESS_READWRITE,
		i_Sub0data := USINT#0,(*Value of subindex0 in array or (def)struct*)
		i_pIndexData := ADR(G_CAN1_VAR.CAN1_RPDO_DUMMY),
		i_itfSDOHandler := DWORD#0
	);
END_IF

(* 16#2130   Application version *)
IF G_CANopen_CAN1_VAR.OD_Error = EPEC_CANopen.Errors.NoError THEN
	G_CANopen_CAN1_VAR.OD_Error := CANopenODAddLine(
		i_pOD := ADR(G_CANopen_CAN1.OD),(*Address of Object dictionary where index will be added*)
		i_index := 16#2130,
		i_ObjectCode := EPEC_CANopen.ObjectCode.OD_ARRAY, (*Type of index*)
		i_NumOfSubids := USINT#10,(*Number of subindexes*)
		i_TypeSpec := EPEC_CANopen.DataType.Deftype_STRING,(*Index of 16-bit deftype*)
		i_ObjectAccess := G_CANOPEN_OD_ACCESS_NOWRITE OR G_CANOPEN_OD_ACCESS_SUB0NOWRITE,
		i_sub0data := USINT#10,(*Value of subindex0 in array or (def)struct*)
		i_pIndexData := ADR(G_SystemInfo.SoftwareInformation),
		i_itfSDOHandler := DWORD#0
	);
END_IF

(* 16#2140   MAC address byte 1 *)
IF G_CANopen_CAN1_VAR.OD_Error = EPEC_CANopen.Errors.NoError THEN
	G_CANopen_CAN1_VAR.OD_Error := CANopenODAddLine(
		i_pOD := ADR(G_CANopen_CAN1.OD),(*Address of Object dictionary where index will be added*)
		i_index := 16#2140,
		i_ObjectCode := EPEC_CANopen.ObjectCode.OD_ARRAY, (*Type of index*)
		i_NumOfSubids := USINT#6,(*Number of subindexes*)
		i_TypeSpec := EPEC_CANopen.DataType.Deftype_UNSIGNED8,(*Index of 16-bit deftype*)
		i_ObjectAccess := G_CANOPEN_OD_ACCESS_NOWRITE OR G_CANOPEN_OD_ACCESS_SUB0NOWRITE,
		i_sub0data := USINT#6,(*Value of subindex0 in array or (def)struct*)
		i_pIndexData := ADR(G_SystemInfo.MACAddress),
		i_itfSDOHandler := DWORD#0
	);
END_IF

(* 16#2141   Ethernet enabled/disabled *)
IF G_CANopen_CAN1_VAR.OD_Error = EPEC_CANopen.Errors.NoError THEN
	G_CANopen_CAN1_VAR.OD_Error := CANopenODAddLine(
		i_pOD := ADR(G_CANopen_CAN1.OD),(*Address of Object dictionary where index will be added*)
		i_index := 16#2141,
		i_ObjectCode := EPEC_CANopen.ObjectCode.OD_ARRAY, (*Type of index*)
		i_NumOfSubids := USINT#50,(*Number of subindexes*)
		i_TypeSpec := EPEC_CANopen.DataType.Deftype_UNSIGNED8,(*Index of 16-bit deftype*)
		i_ObjectAccess := G_CANOPEN_OD_ACCESS_READWRITE OR G_CANOPEN_OD_ACCESS_SUB0NOWRITE,
		i_sub0data := USINT#50,(*Value of subindex0 in array or (def)struct*)
		i_pIndexData := ADR(G_SystemInfo.EthernetConfiguration),
		i_itfSDOHandler := DWORD#0
	);
END_IF

(* 16#2150   CODESYS communication enabled *)
IF G_CANopen_CAN1_VAR.OD_Error = EPEC_CANopen.Errors.NoError THEN
	G_CANopen_CAN1_VAR.OD_Error := CANopenODAddLine(
		i_pOD := ADR(G_CANopen_CAN1.OD),(*Address of Object dictionary where index will be added*)
		i_index := 16#2150,
		i_ObjectCode := EPEC_CANopen.ObjectCode.OD_ARRAY, (*Type of index*)
		i_NumOfSubids := USINT#10,(*Number of subindexes*)
		i_TypeSpec := EPEC_CANopen.DataType.Deftype_UNSIGNED16,(*Index of 16-bit deftype*)
		i_ObjectAccess := G_CANOPEN_OD_ACCESS_READWRITE OR G_CANOPEN_OD_ACCESS_SUB0NOWRITE,
		i_sub0data := USINT#10,(*Value of subindex0 in array or (def)struct*)
		i_pIndexData := ADR(G_SystemInfo.CAN1_Comms),
		i_itfSDOHandler := DWORD#0
	);
END_IF

(* 16#2151   CODESYS communication enabled *)
IF G_CANopen_CAN1_VAR.OD_Error = EPEC_CANopen.Errors.NoError THEN
	G_CANopen_CAN1_VAR.OD_Error := CANopenODAddLine(
		i_pOD := ADR(G_CANopen_CAN1.OD),(*Address of Object dictionary where index will be added*)
		i_index := 16#2151,
		i_ObjectCode := EPEC_CANopen.ObjectCode.OD_ARRAY, (*Type of index*)
		i_NumOfSubids := USINT#10,(*Number of subindexes*)
		i_TypeSpec := EPEC_CANopen.DataType.Deftype_UNSIGNED16,(*Index of 16-bit deftype*)
		i_ObjectAccess := G_CANOPEN_OD_ACCESS_READWRITE OR G_CANOPEN_OD_ACCESS_SUB0NOWRITE,
		i_sub0data := USINT#10,(*Value of subindex0 in array or (def)struct*)
		i_pIndexData := ADR(G_SystemInfo.CAN2_Comms),
		i_itfSDOHandler := DWORD#0
	);
END_IF

(* 16#2152   CODESYS communication enabled *)
IF G_CANopen_CAN1_VAR.OD_Error = EPEC_CANopen.Errors.NoError THEN
	G_CANopen_CAN1_VAR.OD_Error := CANopenODAddLine(
		i_pOD := ADR(G_CANopen_CAN1.OD),(*Address of Object dictionary where index will be added*)
		i_index := 16#2152,
		i_ObjectCode := EPEC_CANopen.ObjectCode.OD_ARRAY, (*Type of index*)
		i_NumOfSubids := USINT#10,(*Number of subindexes*)
		i_TypeSpec := EPEC_CANopen.DataType.Deftype_UNSIGNED16,(*Index of 16-bit deftype*)
		i_ObjectAccess := G_CANOPEN_OD_ACCESS_READWRITE OR G_CANOPEN_OD_ACCESS_SUB0NOWRITE,
		i_sub0data := USINT#10,(*Value of subindex0 in array or (def)struct*)
		i_pIndexData := ADR(G_SystemInfo.CAN3_Comms),
		i_itfSDOHandler := DWORD#0
	);
END_IF

(* 16#2153   CODESYS communication enabled *)
IF G_CANopen_CAN1_VAR.OD_Error = EPEC_CANopen.Errors.NoError THEN
	G_CANopen_CAN1_VAR.OD_Error := CANopenODAddLine(
		i_pOD := ADR(G_CANopen_CAN1.OD),(*Address of Object dictionary where index will be added*)
		i_index := 16#2153,
		i_ObjectCode := EPEC_CANopen.ObjectCode.OD_ARRAY, (*Type of index*)
		i_NumOfSubids := USINT#10,(*Number of subindexes*)
		i_TypeSpec := EPEC_CANopen.DataType.Deftype_UNSIGNED16,(*Index of 16-bit deftype*)
		i_ObjectAccess := G_CANOPEN_OD_ACCESS_READWRITE OR G_CANOPEN_OD_ACCESS_SUB0NOWRITE,
		i_sub0data := USINT#10,(*Value of subindex0 in array or (def)struct*)
		i_pIndexData := ADR(G_SystemInfo.CAN4_Comms),
		i_itfSDOHandler := DWORD#0
	);
END_IF

(* 16#2131 Parameter CSV unique ID *)
IF G_CANopen_CAN1_VAR.OD_Error = EPEC_CANopen.Errors.NoError THEN
	G_CANopen_CAN1_VAR.OD_Error := CANopenODAddLine(
		i_pOD := ADR(G_CANopen_CAN1.OD),(*Address of Object dictionary where index will be added*)
		i_Index := 16#2131,
		i_ObjectCode := EPEC_CANopen.ObjectCode.OD_VAR,(*Type of index*)
		i_NumOfSubids := USINT#0,(*Number of subindexes*)
		i_TypeSpec := EPEC_CANopen.DataType.Deftype_UNSIGNED16,(*Index datatype, either user defined or standard CiA 301*)
		i_ObjectAccess := G_CANOPEN_OD_ACCESS_NOWRITE OR G_CANOPEN_OD_ACCESS_SUB0NOWRITE,
		i_Sub0data := USINT#0,(*Value of subindex0 in array or (def)struct*)
		i_pIndexData := ADR(G_CAN1_VAR.Parameter_CSV_unique_ID1),
		i_itfSDOHandler := DWORD#0
	);
END_IF



G_InitProtocolsCan1State := InitCanProtocolStates.INIT_CANOPEN_PDO;

InitCanProtocolStates.INIT_CANOPEN_PDO:



G_InitProtocolsCan1State := InitCanProtocolStates.INIT_CANOPEN_OD_SAVE;

InitCanProtocolStates.INIT_CANOPEN_OD_SAVE:

(*Initialize OD save*)
G_CANopen_CAN1.SaveAll.Init(i_pParamHandler:=ADR(G_Common.ParHandler));
G_CANopen_CAN1.DeleteAll.Init(i_pParamHandler:=ADR(G_Common.ParHandler));
G_CANopen_CAN1.SaveSubData1010h.pSaveSigns := ADR(G_CANopen_CAN1_VAR.SaveSigns1010[0]);
G_CANopen_CAN1.SaveSubData1010h.NumOfEntrys := 4;
G_CANopen_CAN1.SaveSubData1010h.pSaveIndexData := ADR(G_CANopen_CAN1.SaveData[0]);
G_CANopen_CAN1.SaveData[3].itfSaveAll := G_CANopen_CAN1.SaveAll;
G_CANopen_CAN1.SaveData[3].itfDeleteAll := G_CANopen_CAN1.DeleteAll;
G_CANopen_CAN1.OD.pAdditionalData := ADR(G_CANopen_CAN1.SaveSubData1010h);

IF G_CANopen_CAN1_VAR.OD_Error = EPEC_CANopen.Errors.NoError THEN
	G_CANopen_CAN1.Initialize(i_pOD:=ADR(G_CANopen_CAN1.OD), i_pParamHandler:=ADR(G_Common.ParHandler), o_Error => G_CANopen_CAN1_VAR.ODSave_Error);
END_IF

(* Check all protocol init status flags *)
IF G_CANopen_CAN1_VAR.NMT_Error = EPEC_CANopen.Errors.NoError AND
	G_CANopen_CAN1_VAR.SSDO_Error = EPEC_CANopen.Errors.NoError AND
	G_CANopen_CAN1_VAR.OD_Error = EPEC_CANopen.Errors.NoError AND
	G_CANopen_CAN1_VAR.HB_Error = EPEC_CANopen.Errors.NoError AND
	G_CANopen_CAN1_VAR.CSDO_Error = EPEC_CANopen.Errors.NoError AND
	G_CANopen_CAN1_VAR.GFC_Error = EPEC_CANopen.Errors.NoError
THEN
	G_InitCANopenCan1Error := FALSE; (* No errors in protocol inits *)
ELSE
	G_InitCANopenCan1Error := TRUE;
END_IF



G_InitProtocolsCan1State := InitCanProtocolStates.INIT_J1939;

InitCanProtocolStates.INIT_J1939:

(* AIR1 *)
J1939_CAN1.In.BodyCont.PGN_AIR1.pSPNs:=ADR(J1939_CAN1.In.BodyCont.PGN_AIR1_SPNs);
J1939_CAN1.In.BodyCont.PGN_AIR1.PGN_Number:=16#FEAE;
J1939_CAN1.In.BodyCont.PGN_AIR1.SourceAddress:=16#0021;
J1939_CAN1.In.BodyCont.PGN_AIR1.Destination:=16#00FF;
J1939_CAN1.In.BodyCont.PGN_AIR1.CycleTime:=1000;
J1939_CAN1.In.BodyCont.PGN_AIR1.DataPage:=0;
J1939_CAN1.In.BodyCont.PGN_AIR1.NumberOfSPNs:=7;
J1939_CAN1.In.BodyCont.PGN_AIR1.Priority:=6;
J1939_CAN1.In.BodyCont.PGN_AIR1.DataLength:=7;

	J1939_CAN1.In.BodyCont.PGN_AIR1_SPNs[1].Size:=8; (* BYTE *)
	J1939_CAN1.In.BodyCont.PGN_AIR1_SPNs[1].pData:=ADR(J1939_CAN1.In.BodyCont.AIR1_PneumaticSupplyPress);
	J1939_CAN1.In.BodyCont.PGN_AIR1_SPNs[2].Size:=8; (* BYTE *)
	J1939_CAN1.In.BodyCont.PGN_AIR1_SPNs[2].pData:=ADR(J1939_CAN1.In.BodyCont.AIR1_ParkingAnd_OrTrailerAirPress);
	J1939_CAN1.In.BodyCont.PGN_AIR1_SPNs[3].Size:=8; (* BYTE *)
	J1939_CAN1.In.BodyCont.PGN_AIR1_SPNs[3].pData:=ADR(J1939_CAN1.In.BodyCont.AIR1_ServiceBrakeAirPressCircuit1);
	J1939_CAN1.In.BodyCont.PGN_AIR1_SPNs[4].Size:=8; (* BYTE *)
	J1939_CAN1.In.BodyCont.PGN_AIR1_SPNs[4].pData:=ADR(J1939_CAN1.In.BodyCont.AIR1_ServiceBrakeAirPressCircuit2);
	J1939_CAN1.In.BodyCont.PGN_AIR1_SPNs[5].Size:=8; (* BYTE *)
	J1939_CAN1.In.BodyCont.PGN_AIR1_SPNs[5].pData:=ADR(J1939_CAN1.In.BodyCont.AIR1_AuxEquipmentSupplyPress);
	J1939_CAN1.In.BodyCont.PGN_AIR1_SPNs[6].Size:=8; (* BYTE *)
	J1939_CAN1.In.BodyCont.PGN_AIR1_SPNs[6].pData:=ADR(J1939_CAN1.In.BodyCont.AIR1_AirSuspensionSupplyPress);
	J1939_CAN1.In.BodyCont.PGN_AIR1_SPNs[7].Size:=2; (* BYTE *)
	J1939_CAN1.In.BodyCont.PGN_AIR1_SPNs[7].pData:=ADR(J1939_CAN1.In.BodyCont.AIR1_AirCompressorStatus);
(* EEC2 *)
J1939_CAN1.In.Engine.PGN_EEC2.pSPNs:=ADR(J1939_CAN1.In.Engine.PGN_EEC2_SPNs);
J1939_CAN1.In.Engine.PGN_EEC2.PGN_Number:=16#F003;
J1939_CAN1.In.Engine.PGN_EEC2.SourceAddress:=16#0000;
J1939_CAN1.In.Engine.PGN_EEC2.Destination:=16#00FF;
J1939_CAN1.In.Engine.PGN_EEC2.CycleTime:=50;
J1939_CAN1.In.Engine.PGN_EEC2.DataPage:=0;
J1939_CAN1.In.Engine.PGN_EEC2.NumberOfSPNs:=11;
J1939_CAN1.In.Engine.PGN_EEC2.Priority:=3;
J1939_CAN1.In.Engine.PGN_EEC2.DataLength:=7;

	J1939_CAN1.In.Engine.PGN_EEC2_SPNs[1].Size:=2; (* BYTE *)
	J1939_CAN1.In.Engine.PGN_EEC2_SPNs[1].pData:=ADR(J1939_CAN1.In.Engine.EEC2_AccelPedal1LowIdleSwitch);
	J1939_CAN1.In.Engine.PGN_EEC2_SPNs[2].Size:=2; (* BYTE *)
	J1939_CAN1.In.Engine.PGN_EEC2_SPNs[2].pData:=ADR(J1939_CAN1.In.Engine.EEC2_AccelPedalKickdownSwitch);
	J1939_CAN1.In.Engine.PGN_EEC2_SPNs[3].Size:=2; (* BYTE *)
	J1939_CAN1.In.Engine.PGN_EEC2_SPNs[3].pData:=ADR(J1939_CAN1.In.Engine.EEC2_RoadSpeedLimitStatus);
	J1939_CAN1.In.Engine.PGN_EEC2_SPNs[4].Size:=2; (* BYTE *)
	J1939_CAN1.In.Engine.PGN_EEC2_SPNs[4].pData:=ADR(J1939_CAN1.In.Engine.EEC2_AccelPedal2LowIdleSwitch);
	J1939_CAN1.In.Engine.PGN_EEC2_SPNs[5].Size:=8; (* BYTE *)
	J1939_CAN1.In.Engine.PGN_EEC2_SPNs[5].pData:=ADR(J1939_CAN1.In.Engine.EEC2_AccelPedalPos1);
	J1939_CAN1.In.Engine.PGN_EEC2_SPNs[6].Size:=8; (* BYTE *)
	J1939_CAN1.In.Engine.PGN_EEC2_SPNs[6].pData:=ADR(J1939_CAN1.In.Engine.EEC2_EngPercentLoadAtCurrentSpeed);
	J1939_CAN1.In.Engine.PGN_EEC2_SPNs[7].Size:=8; (* BYTE *)
	J1939_CAN1.In.Engine.PGN_EEC2_SPNs[7].pData:=ADR(J1939_CAN1.In.Engine.EEC2_RemoteAccelPedalPos);
	J1939_CAN1.In.Engine.PGN_EEC2_SPNs[8].Size:=8; (* BYTE *)
	J1939_CAN1.In.Engine.PGN_EEC2_SPNs[8].pData:=ADR(J1939_CAN1.In.Engine.EEC2_AccelPedalPos2);
	J1939_CAN1.In.Engine.PGN_EEC2_SPNs[9].Size:=2; (* BYTE *)
	J1939_CAN1.In.Engine.PGN_EEC2_SPNs[9].pData:=ADR(J1939_CAN1.In.Engine.EEC2_VhclAccelerationRateLimitStatus);
	J1939_CAN1.In.Engine.PGN_EEC2_SPNs[10].Size:=6; (* BYTE *)
	J1939_CAN1.In.Engine.PGN_EEC2_SPNs[10].pData:=ADR(J1939_CAN1.In.Engine.J1939_CAN1_EEC2_Dummy_RX_1);
	J1939_CAN1.In.Engine.PGN_EEC2_SPNs[11].Size:=8; (* BYTE *)
	J1939_CAN1.In.Engine.PGN_EEC2_SPNs[11].pData:=ADR(J1939_CAN1.In.Engine.EEC2_ActMaxAvailEngPercentTorque);
(* CCVS *)
J1939_CAN1.In.CCVS.PGN_CCVS.pSPNs:=ADR(J1939_CAN1.In.CCVS.PGN_CCVS_SPNs);
J1939_CAN1.In.CCVS.PGN_CCVS.PGN_Number:=16#FEF1;
J1939_CAN1.In.CCVS.PGN_CCVS.SourceAddress:=16#0027;
J1939_CAN1.In.CCVS.PGN_CCVS.Destination:=16#00FF;
J1939_CAN1.In.CCVS.PGN_CCVS.CycleTime:=100;
J1939_CAN1.In.CCVS.PGN_CCVS.DataPage:=0;
J1939_CAN1.In.CCVS.PGN_CCVS.NumberOfSPNs:=20;
J1939_CAN1.In.CCVS.PGN_CCVS.Priority:=6;
J1939_CAN1.In.CCVS.PGN_CCVS.DataLength:=8;

	J1939_CAN1.In.CCVS.PGN_CCVS_SPNs[1].Size:=2; (* BYTE *)
	J1939_CAN1.In.CCVS.PGN_CCVS_SPNs[1].pData:=ADR(J1939_CAN1.In.CCVS.CCVS_TwoSpeedAxleSwitch);
	J1939_CAN1.In.CCVS.PGN_CCVS_SPNs[2].Size:=2; (* BYTE *)
	J1939_CAN1.In.CCVS.PGN_CCVS_SPNs[2].pData:=ADR(J1939_CAN1.In.CCVS.CCVS_ParkingBrakeSwitch);
	J1939_CAN1.In.CCVS.PGN_CCVS_SPNs[3].Size:=2; (* BYTE *)
	J1939_CAN1.In.CCVS.PGN_CCVS_SPNs[3].pData:=ADR(J1939_CAN1.In.CCVS.CCVS_CruiseCtrlPauseSwitch);
	J1939_CAN1.In.CCVS.PGN_CCVS_SPNs[4].Size:=2; (* BYTE *)
	J1939_CAN1.In.CCVS.PGN_CCVS_SPNs[4].pData:=ADR(J1939_CAN1.In.CCVS.CCVS_ParkBrakeReleaseInhibitRq);
	J1939_CAN1.In.CCVS.PGN_CCVS_SPNs[5].Size:=16; (* WORD *)
	J1939_CAN1.In.CCVS.PGN_CCVS_SPNs[5].pData:=ADR(J1939_CAN1.In.CCVS.CCVS_WheelBasedVehicleSpeed);
	J1939_CAN1.In.CCVS.PGN_CCVS_SPNs[6].Size:=2; (* BYTE *)
	J1939_CAN1.In.CCVS.PGN_CCVS_SPNs[6].pData:=ADR(J1939_CAN1.In.CCVS.CCVS_CruiseCtrlActive);
	J1939_CAN1.In.CCVS.PGN_CCVS_SPNs[7].Size:=2; (* BYTE *)
	J1939_CAN1.In.CCVS.PGN_CCVS_SPNs[7].pData:=ADR(J1939_CAN1.In.CCVS.CCVS_CruiseCtrlEnableSwitch);
	J1939_CAN1.In.CCVS.PGN_CCVS_SPNs[8].Size:=2; (* BYTE *)
	J1939_CAN1.In.CCVS.PGN_CCVS_SPNs[8].pData:=ADR(J1939_CAN1.In.CCVS.CCVS_BrakeSwitch);
	J1939_CAN1.In.CCVS.PGN_CCVS_SPNs[9].Size:=2; (* BYTE *)
	J1939_CAN1.In.CCVS.PGN_CCVS_SPNs[9].pData:=ADR(J1939_CAN1.In.CCVS.CCVS_ClutchSwitch);
	J1939_CAN1.In.CCVS.PGN_CCVS_SPNs[10].Size:=2; (* BYTE *)
	J1939_CAN1.In.CCVS.PGN_CCVS_SPNs[10].pData:=ADR(J1939_CAN1.In.CCVS.CCVS_CruiseCtrlSetSwitch);
	J1939_CAN1.In.CCVS.PGN_CCVS_SPNs[11].Size:=2; (* BYTE *)
	J1939_CAN1.In.CCVS.PGN_CCVS_SPNs[11].pData:=ADR(J1939_CAN1.In.CCVS.CCVS_CruiseCtrlCoastSwitch);
	J1939_CAN1.In.CCVS.PGN_CCVS_SPNs[12].Size:=2; (* BYTE *)
	J1939_CAN1.In.CCVS.PGN_CCVS_SPNs[12].pData:=ADR(J1939_CAN1.In.CCVS.CCVS_CruiseCtrlResumeSwitch);
	J1939_CAN1.In.CCVS.PGN_CCVS_SPNs[13].Size:=2; (* BYTE *)
	J1939_CAN1.In.CCVS.PGN_CCVS_SPNs[13].pData:=ADR(J1939_CAN1.In.CCVS.CCVS_CruiseCtrlAccelerateSwitch);
	J1939_CAN1.In.CCVS.PGN_CCVS_SPNs[14].Size:=8; (* BYTE *)
	J1939_CAN1.In.CCVS.PGN_CCVS_SPNs[14].pData:=ADR(J1939_CAN1.In.CCVS.CCVS_CruiseCtrlSetSpeed);
	J1939_CAN1.In.CCVS.PGN_CCVS_SPNs[15].Size:=5; (* BYTE *)
	J1939_CAN1.In.CCVS.PGN_CCVS_SPNs[15].pData:=ADR(J1939_CAN1.In.CCVS.CCVS_PTOState);
	J1939_CAN1.In.CCVS.PGN_CCVS_SPNs[16].Size:=3; (* BYTE *)
	J1939_CAN1.In.CCVS.PGN_CCVS_SPNs[16].pData:=ADR(J1939_CAN1.In.CCVS.CCVS_CruiseCtrlStates);
	J1939_CAN1.In.CCVS.PGN_CCVS_SPNs[17].Size:=2; (* BYTE *)
	J1939_CAN1.In.CCVS.PGN_CCVS_SPNs[17].pData:=ADR(J1939_CAN1.In.CCVS.CCVS_EngIdleIncrementSwitch);
	J1939_CAN1.In.CCVS.PGN_CCVS_SPNs[18].Size:=2; (* BYTE *)
	J1939_CAN1.In.CCVS.PGN_CCVS_SPNs[18].pData:=ADR(J1939_CAN1.In.CCVS.CCVS_EngIdleDecrementSwitch);
	J1939_CAN1.In.CCVS.PGN_CCVS_SPNs[19].Size:=2; (* BYTE *)
	J1939_CAN1.In.CCVS.PGN_CCVS_SPNs[19].pData:=ADR(J1939_CAN1.In.CCVS.CCVS_EngTestModeSwitch);
	J1939_CAN1.In.CCVS.PGN_CCVS_SPNs[20].Size:=2; (* BYTE *)
	J1939_CAN1.In.CCVS.PGN_CCVS_SPNs[20].pData:=ADR(J1939_CAN1.In.CCVS.CCVS_EngShutdownOverrideSwitch);

J1939_CAN1.In.PGNs[1].pPGN:=ADR(J1939_CAN1.In.BodyCont.PGN_AIR1);
J1939_CAN1.In.PGNs[2].pPGN:=ADR(J1939_CAN1.In.Engine.PGN_EEC2);
J1939_CAN1.In.PGNs[3].pPGN:=ADR(J1939_CAN1.In.CCVS.PGN_CCVS);

                  
G_InitProtocolsCan1State := InitCanProtocolStates.INIT_PROTOCOLS_DONE;

InitCanProtocolStates.INIT_PROTOCOLS_DONE:
G_InitProtocolsCan1Ready:=TRUE;
END_CASE
END_ACTION

ACTION Init_Protocols_Can2_Action:
(*###########################################################*)
(*This block is created implicit. Don't add own code to here.*)
(*###########################################################*)
;
CASE G_InitProtocolsCan2State OF

InitCanProtocolStates.INIT_CANOPEN_PROTOCOLS:
(*CAN2 INIT*)

G_CANopen_CAN2.Device.itfCanChannel:=G_CAN2_Channel; (*Connect device to can channel*)
G_CANopen_CAN2.Device.NodeID := BYTE#1;
G_CANopen_CAN2.NMT.NmtState:=EPEC_CANopen.NMTState.BootUp; (* Set NMT status to BOOTUP *)

(*Initialize OD's data structures*)
G_CANopen_CAN2.OD.EntryCount:=SIZEOF(G_CANopen_CAN2.ODEntrys)/SIZEOF(G_CANopen_CAN2.ODEntrys[1]); (*Max entries of given OD(CANopenDeviceODEntrys array)*)
G_CANopen_CAN2.OD.InOrder:=FALSE; (*OD isn't in order*)
G_CANopen_CAN2.OD.NextFree:=0; (*OD does not have any entries yet*)
G_CANopen_CAN2.OD.pODEntry:=ADR(G_CANopen_CAN2.ODEntrys); (*Pointer to OD array*)

(*Define NMT protocol*)
G_CANopen_CAN2.Protocols[1].Protocol:=EPEC_CANopen.ProtocolType.NMT;
G_CANopen_CAN2.Protocols[1].pData:=ADR(G_CANopen_CAN2.NMT);
G_CANopen_CAN2.Protocols[1].itfProtocol:=G_CANopen_CAN2.NMT_Handler;
G_CANopen_CAN2.Protocols[1].pError:=ADR(G_CANopen_CAN2_VAR.NMT_Error);
G_CANopen_CAN2_VAR.ProtocolAdded[1] := CANopenDeviceAddProtocol( (* Add to protocol stack *)
	i_pDevice:=ADR(G_CANopen_CAN2.Device),
	i_pProtocol:=ADR(G_CANopen_CAN2.Protocols[1]),
);

(*Initialize NMT protocol*)
IF G_CANopen_CAN2_VAR.ProtocolAdded[1] THEN
	G_CANopen_CAN2.NMT_Handler.Init(
		i_pDevice := ADR(G_CANopen_CAN2.Device),
		i_ThisIsMaster := FALSE,
		i_StartInterval :=  1000,
		i_pMonitoredNodes := 0,
		i_NumberOfNodes := 0,
		i_SimultaneousSlaveConfiguration := FALSE,
		o_Error => G_CANopen_CAN2_VAR.NMT_Error
	);
ELSE
	G_CANopen_CAN2_VAR.NMT_Error := EPEC_CANopen.Errors.ProtocolDataMissing;
END_IF

(*Define OD protocol*)
G_CANopen_CAN2.Protocols[2].Protocol:=EPEC_CANopen.ProtocolType.OD;
G_CANopen_CAN2.Protocols[2].pData:=ADR(G_CANopen_CAN2.OD);
G_CANopen_CAN2.Protocols[2].pError:=ADR(G_CANopen_CAN2_VAR.OD_Error);
G_CANopen_CAN2_VAR.ProtocolAdded[2] := CANopenDeviceAddProtocol( (* Add to protocol stack *)
	i_pDevice:=ADR(G_CANopen_CAN2.Device),
	i_pProtocol:=ADR(G_CANopen_CAN2.Protocols[2]),
);
IF NOT G_CANopen_CAN2_VAR.ProtocolAdded[2] THEN
	G_CANopen_CAN2_VAR.OD_Error := EPEC_CANopen.Errors.ProtocolDataMissing;
END_IF

(*Define HB protocol
- Uses NMT and OD protocol data, thus need to be defined after them.
*)
G_CANopen_CAN2.HB.HeartBeat.PT := T#200MS; (* HB producer time *)

G_CANopen_CAN2.Protocols[3].Protocol:=EPEC_CANopen.ProtocolType.HB;
G_CANopen_CAN2.Protocols[3].pData:=ADR(G_CANopen_CAN2.HB);
G_CANopen_CAN2.Protocols[3].itfProtocol:=G_CANopen_CAN2.HB_Handler;
G_CANopen_CAN2.Protocols[3].pError:=ADR(G_CANopen_CAN2_VAR.HB_Error);
G_CANopen_CAN2_VAR.ProtocolAdded[3] := CANopenDeviceAddProtocol( (* Add to protocol stack *)
	i_pDevice:=ADR(G_CANopen_CAN2.Device),
	i_pProtocol:=ADR(G_CANopen_CAN2.Protocols[3]),
);

(* Initialize HB protocol *)
IF G_CANopen_CAN2_VAR.ProtocolAdded[3] THEN
	G_CANopen_CAN2.HB_Handler.Init(
		i_pDevice := ADR(G_CANopen_CAN2.Device),
		o_Error => G_CANopen_CAN2_VAR.HB_Error
	);

	(* Add monitored nodes *)
ELSE
	G_CANopen_CAN2_VAR.HB_Error := EPEC_CANopen.Errors.ProtocolDataMissing;
END_IF

(*Define SSDO protocol*)
G_CANopen_CAN2.Protocols[4].Protocol:=EPEC_CANopen.ProtocolType.SSDO;
G_CANopen_CAN2.Protocols[4].pData:=ADR(G_CANopen_CAN2.SSDO);
G_CANopen_CAN2.Protocols[4].itfProtocol:=G_CANopen_CAN2.SSDO_Handler;
G_CANopen_CAN2.Protocols[4].pError:=ADR(G_CANopen_CAN2_VAR.SSDO_Error);
G_CANopen_CAN2_VAR.ProtocolAdded[4] := CANopenDeviceAddProtocol( (* Add to protocol stack *)
	i_pDevice:=ADR(G_CANopen_CAN2.Device),
	i_pProtocol:=ADR(G_CANopen_CAN2.Protocols[4])
);
IF G_CANopen_CAN2_VAR.ProtocolAdded[4] THEN
	G_CANopen_CAN2.SSDO_Handler.Init(
		i_pDevice := ADR(G_CANopen_CAN2.Device),
		o_Error => G_CANopen_CAN2_VAR.SSDO_Error
	);
ELSE
	G_CANopen_CAN2_VAR.SSDO_Error := EPEC_CANopen.Errors.ProtocolDataMissing;
END_IF

(*Define GFC protocol*)
G_CANopen_CAN2.Protocols[5].Protocol:=EPEC_CANopen.ProtocolType.GFC;
G_CANopen_CAN2.Protocols[5].pData:=ADR(G_CANopen_CAN2.GFC);
G_CANopen_CAN2.Protocols[5].itfProtocol:=G_CANopen_CAN2.GFC_Handler;
G_CANopen_CAN2.Protocols[5].pError:=ADR(G_CANopen_CAN2_VAR.GFC_Error);
G_CANopen_CAN2_VAR.ProtocolAdded[5] := CANopenDeviceAddProtocol(  (* Add to protocol stack *)
	i_pDevice:=ADR(G_CANopen_CAN2.Device),
	i_pProtocol:=ADR(G_CANopen_CAN2.Protocols[5])
);
IF G_CANopen_CAN2_VAR.ProtocolAdded[5] THEN
	G_CANopen_CAN2.GFC_Handler.Init(
		i_pDevice := ADR(G_CANopen_CAN2.Device),
		i_pStatus:=ADR(G_CANopen_CAN2_VAR.GFC_Status),
		o_Error => G_CANopen_CAN2_VAR.GFC_Error
	);
ELSE
	G_CANopen_CAN2_VAR.GFC_Error := EPEC_CANopen.Errors.ProtocolDataMissing;
END_IF

(* Init CSDO instance array for bus *)
EPEC_CANopen.CANopenSDOManager.Init(
	i_pDevice:=ADR(G_CANopen_CAN2.Device),
	i_NodeId:=G_CANopen_CAN2.Device.NodeID,
	i_pCsdoArrayStart:=ADR(G_CANopen_CAN2.CSDOS),
	i_CsdoArraySize:=127,
	o_Error=>G_CANopen_CAN2_VAR.CSDO_Error
);





G_InitProtocolsCan2State := InitCanProtocolStates.INIT_CANOPEN_OD;

InitCanProtocolStates.INIT_CANOPEN_OD:

(*16#0001..16#0009 Default types *)
G_CANopen_CAN2_VAR.OD_Error := EPEC_CANopen.CANopenODAddDefautTypes(
	i_pOD:= ADR(G_CANopen_CAN2.OD)
);

(* 16#1000 Information about the device type *)
IF G_CANopen_CAN2_VAR.OD_Error = EPEC_CANopen.Errors.NoError THEN
	G_CANopen_CAN2_VAR.OD_Error := CANopenODAddLine(
		i_pOD := ADR(G_CANopen_CAN2.OD),(*Address of Object dictionary where index will be added*)
		i_Index := G_CANOPEN_ODINDEX_DEVICE_TYPE,
		i_ObjectCode := EPEC_CANopen.ObjectCode.OD_VAR,(*Type of index*)
		i_NumOfSubids := USINT#0,(*Number of subindexes*)
		i_TypeSpec := EPEC_CANopen.DataType.Deftype_UNSIGNED32,(*Index datatype, either user defined or standard CiA 301*)
		i_ObjectAccess := G_CANOPEN_OD_ACCESS_NOWRITE OR G_CANOPEN_OD_ACCESS_SUB0NOWRITE,
		i_Sub0data := USINT#0,(*Value of subindex0 in array or (def)struct*)
		i_pIndexData := ADR(G_CAN2_VAR.DeviceType_Device2),
		i_itfSDOHandler := DWORD#0
	);
END_IF

(* 16#1001 Error information *)
IF G_CANopen_CAN2_VAR.OD_Error = EPEC_CANopen.Errors.NoError THEN
	G_CANopen_CAN2_VAR.OD_Error := CANopenODAddLine(
		i_pOD := ADR(G_CANopen_CAN2.OD),(*Address of Object dictionary where index will be added*)
		i_Index := G_CANOPEN_ODINDEX_ERROR_REGISTER,
		i_ObjectCode := EPEC_CANopen.ObjectCode.OD_VAR,(*Type of index*)
		i_NumOfSubids := USINT#0,(*Number of subindexes*)
		i_TypeSpec := EPEC_CANopen.DataType.Deftype_UNSIGNED8,(*Index datatype, either user defined or standard CiA 301*)
		i_ObjectAccess := G_CANOPEN_OD_ACCESS_NOWRITE OR G_CANOPEN_OD_ACCESS_SUB0NOWRITE,
		i_Sub0data := USINT#0,(*Value of subindex0 in array or (def)struct*)
		i_pIndexData := ADR(G_CAN2_VAR.ErrorReg_Device2),
		i_itfSDOHandler := DWORD#0
	);
END_IF

(* 16#100A Manufacturer software version *)
IF G_CANopen_CAN2_VAR.OD_Error = EPEC_CANopen.Errors.NoError THEN
	G_CANopen_CAN2_VAR.OD_Error := CANopenODAddLine(
		i_pOD := ADR(G_CANopen_CAN2.OD),(*Address of Object dictionary where index will be added*)
		i_Index := G_CANOPEN_ODINDEX_MF_SW_VERSION,
		i_ObjectCode := EPEC_CANopen.ObjectCode.OD_VAR,(*Type of index*)
		i_NumOfSubids := USINT#0,(*Number of subindexes*)
		i_TypeSpec := EPEC_CANopen.DataType.Deftype_STRING,(*Index datatype, either user defined or standard CiA 301*)
		i_ObjectAccess := G_CANOPEN_OD_ACCESS_NOWRITE OR G_CANOPEN_OD_ACCESS_SUB0NOWRITE,
		i_Sub0data := USINT#0,(*Value of subindex0 in array or (def)struct*)
		i_pIndexData := ADR(G_SystemInfo.SWVersion),
		i_itfSDOHandler := DWORD#0
	);
END_IF

(* 16#1018   Vendor ID *)
IF G_CANopen_CAN2_VAR.OD_Error = EPEC_CANopen.Errors.NoError THEN
	G_CANopen_CAN2_VAR.OD_Error := CANopenODAddLine(
		i_pOD := ADR(G_CANopen_CAN2.OD),(*Address of Object dictionary where index will be added*)
		i_index := G_CANOPEN_ODINDEX_IDENTITY_OBJECT,
		i_ObjectCode := EPEC_CANopen.ObjectCode.OD_ARRAY, (*Type of index*)
		i_NumOfSubids := USINT#4,(*Number of subindexes*)
		i_TypeSpec := EPEC_CANopen.DataType.Deftype_UNSIGNED32,(*Index of 16-bit deftype*)
		i_ObjectAccess := G_CANOPEN_OD_ACCESS_NOWRITE OR G_CANOPEN_OD_ACCESS_SUB0NOWRITE,
		i_sub0data := USINT#4,(*Value of subindex0 in array or (def)struct*)
		i_pIndexData := ADR(G_SystemInfo.Identity),
		i_itfSDOHandler := DWORD#0
	);
END_IF
(* 16#2128 PDO Dummy Variable Index *)
IF G_CANopen_CAN2_VAR.OD_Error = EPEC_CANopen.Errors.NoError THEN
	G_CANopen_CAN2_VAR.OD_Error := CANopenODAddLine(
		i_pOD := ADR(G_CANopen_CAN2.OD),(*Address of Object dictionary where index will be added*)
		i_Index := 16#2128,
		i_ObjectCode := EPEC_CANopen.ObjectCode.OD_VAR,(*Type of index*)
		i_NumOfSubids := USINT#0,(*Number of subindexes*)
		i_TypeSpec := EPEC_CANopen.DataType.Deftype_UNSIGNED8,(*Index datatype, either user defined or standard CiA 301*)
		i_ObjectAccess := G_CANOPEN_OD_ACCESS_READWRITE,
		i_Sub0data := USINT#0,(*Value of subindex0 in array or (def)struct*)
		i_pIndexData := ADR(G_CAN2_VAR.CAN2_TPDO_DUMMY),
		i_itfSDOHandler := DWORD#0
	);
END_IF

(* 16#2129 PDO Dummy Variable Index *)
IF G_CANopen_CAN2_VAR.OD_Error = EPEC_CANopen.Errors.NoError THEN
	G_CANopen_CAN2_VAR.OD_Error := CANopenODAddLine(
		i_pOD := ADR(G_CANopen_CAN2.OD),(*Address of Object dictionary where index will be added*)
		i_Index := 16#2129,
		i_ObjectCode := EPEC_CANopen.ObjectCode.OD_VAR,(*Type of index*)
		i_NumOfSubids := USINT#0,(*Number of subindexes*)
		i_TypeSpec := EPEC_CANopen.DataType.Deftype_UNSIGNED8,(*Index datatype, either user defined or standard CiA 301*)
		i_ObjectAccess := G_CANOPEN_OD_ACCESS_READWRITE,
		i_Sub0data := USINT#0,(*Value of subindex0 in array or (def)struct*)
		i_pIndexData := ADR(G_CAN2_VAR.CAN2_RPDO_DUMMY),
		i_itfSDOHandler := DWORD#0
	);
END_IF

(* 16#2130   Application version *)
IF G_CANopen_CAN2_VAR.OD_Error = EPEC_CANopen.Errors.NoError THEN
	G_CANopen_CAN2_VAR.OD_Error := CANopenODAddLine(
		i_pOD := ADR(G_CANopen_CAN2.OD),(*Address of Object dictionary where index will be added*)
		i_index := 16#2130,
		i_ObjectCode := EPEC_CANopen.ObjectCode.OD_ARRAY, (*Type of index*)
		i_NumOfSubids := USINT#10,(*Number of subindexes*)
		i_TypeSpec := EPEC_CANopen.DataType.Deftype_STRING,(*Index of 16-bit deftype*)
		i_ObjectAccess := G_CANOPEN_OD_ACCESS_NOWRITE OR G_CANOPEN_OD_ACCESS_SUB0NOWRITE,
		i_sub0data := USINT#10,(*Value of subindex0 in array or (def)struct*)
		i_pIndexData := ADR(G_SystemInfo.SoftwareInformation),
		i_itfSDOHandler := DWORD#0
	);
END_IF

(* 16#2131 Parameter CSV unique ID *)
IF G_CANopen_CAN2_VAR.OD_Error = EPEC_CANopen.Errors.NoError THEN
	G_CANopen_CAN2_VAR.OD_Error := CANopenODAddLine(
		i_pOD := ADR(G_CANopen_CAN2.OD),(*Address of Object dictionary where index will be added*)
		i_Index := 16#2131,
		i_ObjectCode := EPEC_CANopen.ObjectCode.OD_VAR,(*Type of index*)
		i_NumOfSubids := USINT#0,(*Number of subindexes*)
		i_TypeSpec := EPEC_CANopen.DataType.Deftype_UNSIGNED16,(*Index datatype, either user defined or standard CiA 301*)
		i_ObjectAccess := G_CANOPEN_OD_ACCESS_NOWRITE OR G_CANOPEN_OD_ACCESS_SUB0NOWRITE,
		i_Sub0data := USINT#0,(*Value of subindex0 in array or (def)struct*)
		i_pIndexData := ADR(G_CAN2_VAR.Parameter_CSV_unique_ID2),
		i_itfSDOHandler := DWORD#0
	);
END_IF



G_InitProtocolsCan2State := InitCanProtocolStates.INIT_CANOPEN_PDO;

InitCanProtocolStates.INIT_CANOPEN_PDO:



G_InitProtocolsCan2State := InitCanProtocolStates.INIT_CANOPEN_OD_SAVE;

InitCanProtocolStates.INIT_CANOPEN_OD_SAVE:

(*Initialize OD save*)
G_CANopen_CAN2.SaveAll.Init(i_pParamHandler:=ADR(G_Common.ParHandler));
G_CANopen_CAN2.DeleteAll.Init(i_pParamHandler:=ADR(G_Common.ParHandler));
G_CANopen_CAN2.SaveSubData1010h.pSaveSigns := ADR(G_CANopen_CAN2_VAR.SaveSigns1010[0]);
G_CANopen_CAN2.SaveSubData1010h.NumOfEntrys := 4;
G_CANopen_CAN2.SaveSubData1010h.pSaveIndexData := ADR(G_CANopen_CAN2.SaveData[0]);
G_CANopen_CAN2.SaveData[3].itfSaveAll := G_CANopen_CAN2.SaveAll;
G_CANopen_CAN2.SaveData[3].itfDeleteAll := G_CANopen_CAN2.DeleteAll;
G_CANopen_CAN2.OD.pAdditionalData := ADR(G_CANopen_CAN2.SaveSubData1010h);

IF G_CANopen_CAN2_VAR.OD_Error = EPEC_CANopen.Errors.NoError THEN
	G_CANopen_CAN2.Initialize(i_pOD:=ADR(G_CANopen_CAN2.OD), i_pParamHandler:=ADR(G_Common.ParHandler), o_Error => G_CANopen_CAN2_VAR.ODSave_Error);
END_IF

(* Check all protocol init status flags *)
IF G_CANopen_CAN2_VAR.NMT_Error = EPEC_CANopen.Errors.NoError AND
	G_CANopen_CAN2_VAR.SSDO_Error = EPEC_CANopen.Errors.NoError AND
	G_CANopen_CAN2_VAR.OD_Error = EPEC_CANopen.Errors.NoError AND
	G_CANopen_CAN2_VAR.HB_Error = EPEC_CANopen.Errors.NoError AND
	G_CANopen_CAN2_VAR.CSDO_Error = EPEC_CANopen.Errors.NoError AND
	G_CANopen_CAN2_VAR.GFC_Error = EPEC_CANopen.Errors.NoError
THEN
	G_InitCANopenCan2Error := FALSE; (* No errors in protocol inits *)
ELSE
	G_InitCANopenCan2Error := TRUE;
END_IF



G_InitProtocolsCan2State := InitCanProtocolStates.INIT_J1939;

InitCanProtocolStates.INIT_J1939:



                  
G_InitProtocolsCan2State := InitCanProtocolStates.INIT_PROTOCOLS_DONE;

InitCanProtocolStates.INIT_PROTOCOLS_DONE:
G_InitProtocolsCan2Ready:=TRUE;
END_CASE
END_ACTION

ACTION Init_Protocols_Can3_Action:
(*###########################################################*)
(*This block is created implicit. Don't add own code to here.*)
(*###########################################################*)
;
CASE G_InitProtocolsCan3State OF

InitCanProtocolStates.INIT_CANOPEN_PROTOCOLS:
(*CAN3 INIT*)

G_CANopen_CAN3.Device.itfCanChannel:=G_CAN3_Channel; (*Connect device to can channel*)
G_CANopen_CAN3.Device.NodeID := BYTE#1;
G_CANopen_CAN3.NMT.NmtState:=EPEC_CANopen.NMTState.BootUp; (* Set NMT status to BOOTUP *)

(*Initialize OD's data structures*)
G_CANopen_CAN3.OD.EntryCount:=SIZEOF(G_CANopen_CAN3.ODEntrys)/SIZEOF(G_CANopen_CAN3.ODEntrys[1]); (*Max entries of given OD(CANopenDeviceODEntrys array)*)
G_CANopen_CAN3.OD.InOrder:=FALSE; (*OD isn't in order*)
G_CANopen_CAN3.OD.NextFree:=0; (*OD does not have any entries yet*)
G_CANopen_CAN3.OD.pODEntry:=ADR(G_CANopen_CAN3.ODEntrys); (*Pointer to OD array*)

(*Define NMT protocol*)
G_CANopen_CAN3.Protocols[1].Protocol:=EPEC_CANopen.ProtocolType.NMT;
G_CANopen_CAN3.Protocols[1].pData:=ADR(G_CANopen_CAN3.NMT);
G_CANopen_CAN3.Protocols[1].itfProtocol:=G_CANopen_CAN3.NMT_Handler;
G_CANopen_CAN3.Protocols[1].pError:=ADR(G_CANopen_CAN3_VAR.NMT_Error);
G_CANopen_CAN3_VAR.ProtocolAdded[1] := CANopenDeviceAddProtocol( (* Add to protocol stack *)
	i_pDevice:=ADR(G_CANopen_CAN3.Device),
	i_pProtocol:=ADR(G_CANopen_CAN3.Protocols[1]),
);

(*Initialize NMT protocol*)
IF G_CANopen_CAN3_VAR.ProtocolAdded[1] THEN
	G_CANopen_CAN3.NMT_Handler.Init(
		i_pDevice := ADR(G_CANopen_CAN3.Device),
		i_ThisIsMaster := FALSE,
		i_StartInterval :=  1000,
		i_pMonitoredNodes := 0,
		i_NumberOfNodes := 0,
		i_SimultaneousSlaveConfiguration := FALSE,
		o_Error => G_CANopen_CAN3_VAR.NMT_Error
	);
ELSE
	G_CANopen_CAN3_VAR.NMT_Error := EPEC_CANopen.Errors.ProtocolDataMissing;
END_IF

(*Define OD protocol*)
G_CANopen_CAN3.Protocols[2].Protocol:=EPEC_CANopen.ProtocolType.OD;
G_CANopen_CAN3.Protocols[2].pData:=ADR(G_CANopen_CAN3.OD);
G_CANopen_CAN3.Protocols[2].pError:=ADR(G_CANopen_CAN3_VAR.OD_Error);
G_CANopen_CAN3_VAR.ProtocolAdded[2] := CANopenDeviceAddProtocol( (* Add to protocol stack *)
	i_pDevice:=ADR(G_CANopen_CAN3.Device),
	i_pProtocol:=ADR(G_CANopen_CAN3.Protocols[2]),
);
IF NOT G_CANopen_CAN3_VAR.ProtocolAdded[2] THEN
	G_CANopen_CAN3_VAR.OD_Error := EPEC_CANopen.Errors.ProtocolDataMissing;
END_IF

(*Define HB protocol
- Uses NMT and OD protocol data, thus need to be defined after them.
*)
G_CANopen_CAN3.HB.HeartBeat.PT := T#200MS; (* HB producer time *)

G_CANopen_CAN3.Protocols[3].Protocol:=EPEC_CANopen.ProtocolType.HB;
G_CANopen_CAN3.Protocols[3].pData:=ADR(G_CANopen_CAN3.HB);
G_CANopen_CAN3.Protocols[3].itfProtocol:=G_CANopen_CAN3.HB_Handler;
G_CANopen_CAN3.Protocols[3].pError:=ADR(G_CANopen_CAN3_VAR.HB_Error);
G_CANopen_CAN3_VAR.ProtocolAdded[3] := CANopenDeviceAddProtocol( (* Add to protocol stack *)
	i_pDevice:=ADR(G_CANopen_CAN3.Device),
	i_pProtocol:=ADR(G_CANopen_CAN3.Protocols[3]),
);

(* Initialize HB protocol *)
IF G_CANopen_CAN3_VAR.ProtocolAdded[3] THEN
	G_CANopen_CAN3.HB_Handler.Init(
		i_pDevice := ADR(G_CANopen_CAN3.Device),
		o_Error => G_CANopen_CAN3_VAR.HB_Error
	);

	(* Add monitored nodes *)
ELSE
	G_CANopen_CAN3_VAR.HB_Error := EPEC_CANopen.Errors.ProtocolDataMissing;
END_IF

(*Define SSDO protocol*)
G_CANopen_CAN3.Protocols[4].Protocol:=EPEC_CANopen.ProtocolType.SSDO;
G_CANopen_CAN3.Protocols[4].pData:=ADR(G_CANopen_CAN3.SSDO);
G_CANopen_CAN3.Protocols[4].itfProtocol:=G_CANopen_CAN3.SSDO_Handler;
G_CANopen_CAN3.Protocols[4].pError:=ADR(G_CANopen_CAN3_VAR.SSDO_Error);
G_CANopen_CAN3_VAR.ProtocolAdded[4] := CANopenDeviceAddProtocol( (* Add to protocol stack *)
	i_pDevice:=ADR(G_CANopen_CAN3.Device),
	i_pProtocol:=ADR(G_CANopen_CAN3.Protocols[4])
);
IF G_CANopen_CAN3_VAR.ProtocolAdded[4] THEN
	G_CANopen_CAN3.SSDO_Handler.Init(
		i_pDevice := ADR(G_CANopen_CAN3.Device),
		o_Error => G_CANopen_CAN3_VAR.SSDO_Error
	);
ELSE
	G_CANopen_CAN3_VAR.SSDO_Error := EPEC_CANopen.Errors.ProtocolDataMissing;
END_IF

(*Define GFC protocol*)
G_CANopen_CAN3.Protocols[5].Protocol:=EPEC_CANopen.ProtocolType.GFC;
G_CANopen_CAN3.Protocols[5].pData:=ADR(G_CANopen_CAN3.GFC);
G_CANopen_CAN3.Protocols[5].itfProtocol:=G_CANopen_CAN3.GFC_Handler;
G_CANopen_CAN3.Protocols[5].pError:=ADR(G_CANopen_CAN3_VAR.GFC_Error);
G_CANopen_CAN3_VAR.ProtocolAdded[5] := CANopenDeviceAddProtocol(  (* Add to protocol stack *)
	i_pDevice:=ADR(G_CANopen_CAN3.Device),
	i_pProtocol:=ADR(G_CANopen_CAN3.Protocols[5])
);
IF G_CANopen_CAN3_VAR.ProtocolAdded[5] THEN
	G_CANopen_CAN3.GFC_Handler.Init(
		i_pDevice := ADR(G_CANopen_CAN3.Device),
		i_pStatus:=ADR(G_CANopen_CAN3_VAR.GFC_Status),
		o_Error => G_CANopen_CAN3_VAR.GFC_Error
	);
ELSE
	G_CANopen_CAN3_VAR.GFC_Error := EPEC_CANopen.Errors.ProtocolDataMissing;
END_IF

(* Init CSDO instance array for bus *)
EPEC_CANopen.CANopenSDOManager.Init(
	i_pDevice:=ADR(G_CANopen_CAN3.Device),
	i_NodeId:=G_CANopen_CAN3.Device.NodeID,
	i_pCsdoArrayStart:=ADR(G_CANopen_CAN3.CSDOS),
	i_CsdoArraySize:=127,
	o_Error=>G_CANopen_CAN3_VAR.CSDO_Error
);





G_InitProtocolsCan3State := InitCanProtocolStates.INIT_CANOPEN_OD;

InitCanProtocolStates.INIT_CANOPEN_OD:

(*16#0001..16#0009 Default types *)
G_CANopen_CAN3_VAR.OD_Error := EPEC_CANopen.CANopenODAddDefautTypes(
	i_pOD:= ADR(G_CANopen_CAN3.OD)
);

(* 16#1000 Information about the device type *)
IF G_CANopen_CAN3_VAR.OD_Error = EPEC_CANopen.Errors.NoError THEN
	G_CANopen_CAN3_VAR.OD_Error := CANopenODAddLine(
		i_pOD := ADR(G_CANopen_CAN3.OD),(*Address of Object dictionary where index will be added*)
		i_Index := G_CANOPEN_ODINDEX_DEVICE_TYPE,
		i_ObjectCode := EPEC_CANopen.ObjectCode.OD_VAR,(*Type of index*)
		i_NumOfSubids := USINT#0,(*Number of subindexes*)
		i_TypeSpec := EPEC_CANopen.DataType.Deftype_UNSIGNED32,(*Index datatype, either user defined or standard CiA 301*)
		i_ObjectAccess := G_CANOPEN_OD_ACCESS_NOWRITE OR G_CANOPEN_OD_ACCESS_SUB0NOWRITE,
		i_Sub0data := USINT#0,(*Value of subindex0 in array or (def)struct*)
		i_pIndexData := ADR(G_CAN3_VAR.DeviceType_Device3),
		i_itfSDOHandler := DWORD#0
	);
END_IF

(* 16#1001 Error information *)
IF G_CANopen_CAN3_VAR.OD_Error = EPEC_CANopen.Errors.NoError THEN
	G_CANopen_CAN3_VAR.OD_Error := CANopenODAddLine(
		i_pOD := ADR(G_CANopen_CAN3.OD),(*Address of Object dictionary where index will be added*)
		i_Index := G_CANOPEN_ODINDEX_ERROR_REGISTER,
		i_ObjectCode := EPEC_CANopen.ObjectCode.OD_VAR,(*Type of index*)
		i_NumOfSubids := USINT#0,(*Number of subindexes*)
		i_TypeSpec := EPEC_CANopen.DataType.Deftype_UNSIGNED8,(*Index datatype, either user defined or standard CiA 301*)
		i_ObjectAccess := G_CANOPEN_OD_ACCESS_NOWRITE OR G_CANOPEN_OD_ACCESS_SUB0NOWRITE,
		i_Sub0data := USINT#0,(*Value of subindex0 in array or (def)struct*)
		i_pIndexData := ADR(G_CAN3_VAR.ErrorReg_Device3),
		i_itfSDOHandler := DWORD#0
	);
END_IF

(* 16#100A Manufacturer software version *)
IF G_CANopen_CAN3_VAR.OD_Error = EPEC_CANopen.Errors.NoError THEN
	G_CANopen_CAN3_VAR.OD_Error := CANopenODAddLine(
		i_pOD := ADR(G_CANopen_CAN3.OD),(*Address of Object dictionary where index will be added*)
		i_Index := G_CANOPEN_ODINDEX_MF_SW_VERSION,
		i_ObjectCode := EPEC_CANopen.ObjectCode.OD_VAR,(*Type of index*)
		i_NumOfSubids := USINT#0,(*Number of subindexes*)
		i_TypeSpec := EPEC_CANopen.DataType.Deftype_STRING,(*Index datatype, either user defined or standard CiA 301*)
		i_ObjectAccess := G_CANOPEN_OD_ACCESS_NOWRITE OR G_CANOPEN_OD_ACCESS_SUB0NOWRITE,
		i_Sub0data := USINT#0,(*Value of subindex0 in array or (def)struct*)
		i_pIndexData := ADR(G_SystemInfo.SWVersion),
		i_itfSDOHandler := DWORD#0
	);
END_IF

(* 16#1018   Vendor ID *)
IF G_CANopen_CAN3_VAR.OD_Error = EPEC_CANopen.Errors.NoError THEN
	G_CANopen_CAN3_VAR.OD_Error := CANopenODAddLine(
		i_pOD := ADR(G_CANopen_CAN3.OD),(*Address of Object dictionary where index will be added*)
		i_index := G_CANOPEN_ODINDEX_IDENTITY_OBJECT,
		i_ObjectCode := EPEC_CANopen.ObjectCode.OD_ARRAY, (*Type of index*)
		i_NumOfSubids := USINT#4,(*Number of subindexes*)
		i_TypeSpec := EPEC_CANopen.DataType.Deftype_UNSIGNED32,(*Index of 16-bit deftype*)
		i_ObjectAccess := G_CANOPEN_OD_ACCESS_NOWRITE OR G_CANOPEN_OD_ACCESS_SUB0NOWRITE,
		i_sub0data := USINT#4,(*Value of subindex0 in array or (def)struct*)
		i_pIndexData := ADR(G_SystemInfo.Identity),
		i_itfSDOHandler := DWORD#0
	);
END_IF
(* 16#2129 PDO Dummy Variable Index *)
IF G_CANopen_CAN3_VAR.OD_Error = EPEC_CANopen.Errors.NoError THEN
	G_CANopen_CAN3_VAR.OD_Error := CANopenODAddLine(
		i_pOD := ADR(G_CANopen_CAN3.OD),(*Address of Object dictionary where index will be added*)
		i_Index := 16#2129,
		i_ObjectCode := EPEC_CANopen.ObjectCode.OD_VAR,(*Type of index*)
		i_NumOfSubids := USINT#0,(*Number of subindexes*)
		i_TypeSpec := EPEC_CANopen.DataType.Deftype_UNSIGNED8,(*Index datatype, either user defined or standard CiA 301*)
		i_ObjectAccess := G_CANOPEN_OD_ACCESS_READWRITE,
		i_Sub0data := USINT#0,(*Value of subindex0 in array or (def)struct*)
		i_pIndexData := ADR(G_CAN3_VAR.CAN3_PDO_DUMMY),
		i_itfSDOHandler := DWORD#0
	);
END_IF

(* 16#2130   Application version *)
IF G_CANopen_CAN3_VAR.OD_Error = EPEC_CANopen.Errors.NoError THEN
	G_CANopen_CAN3_VAR.OD_Error := CANopenODAddLine(
		i_pOD := ADR(G_CANopen_CAN3.OD),(*Address of Object dictionary where index will be added*)
		i_index := 16#2130,
		i_ObjectCode := EPEC_CANopen.ObjectCode.OD_ARRAY, (*Type of index*)
		i_NumOfSubids := USINT#10,(*Number of subindexes*)
		i_TypeSpec := EPEC_CANopen.DataType.Deftype_STRING,(*Index of 16-bit deftype*)
		i_ObjectAccess := G_CANOPEN_OD_ACCESS_NOWRITE OR G_CANOPEN_OD_ACCESS_SUB0NOWRITE,
		i_sub0data := USINT#10,(*Value of subindex0 in array or (def)struct*)
		i_pIndexData := ADR(G_SystemInfo.SoftwareInformation),
		i_itfSDOHandler := DWORD#0
	);
END_IF

(* 16#2131 Parameter CSV unique ID *)
IF G_CANopen_CAN3_VAR.OD_Error = EPEC_CANopen.Errors.NoError THEN
	G_CANopen_CAN3_VAR.OD_Error := CANopenODAddLine(
		i_pOD := ADR(G_CANopen_CAN3.OD),(*Address of Object dictionary where index will be added*)
		i_Index := 16#2131,
		i_ObjectCode := EPEC_CANopen.ObjectCode.OD_VAR,(*Type of index*)
		i_NumOfSubids := USINT#0,(*Number of subindexes*)
		i_TypeSpec := EPEC_CANopen.DataType.Deftype_UNSIGNED16,(*Index datatype, either user defined or standard CiA 301*)
		i_ObjectAccess := G_CANOPEN_OD_ACCESS_NOWRITE OR G_CANOPEN_OD_ACCESS_SUB0NOWRITE,
		i_Sub0data := USINT#0,(*Value of subindex0 in array or (def)struct*)
		i_pIndexData := ADR(G_CAN3_VAR.Parameter_CSV_unique_ID3),
		i_itfSDOHandler := DWORD#0
	);
END_IF



G_InitProtocolsCan3State := InitCanProtocolStates.INIT_CANOPEN_PDO;

InitCanProtocolStates.INIT_CANOPEN_PDO:



G_InitProtocolsCan3State := InitCanProtocolStates.INIT_CANOPEN_OD_SAVE;

InitCanProtocolStates.INIT_CANOPEN_OD_SAVE:

(*Initialize OD save*)
G_CANopen_CAN3.SaveAll.Init(i_pParamHandler:=ADR(G_Common.ParHandler));
G_CANopen_CAN3.DeleteAll.Init(i_pParamHandler:=ADR(G_Common.ParHandler));
G_CANopen_CAN3.SaveSubData1010h.pSaveSigns := ADR(G_CANopen_CAN3_VAR.SaveSigns1010[0]);
G_CANopen_CAN3.SaveSubData1010h.NumOfEntrys := 4;
G_CANopen_CAN3.SaveSubData1010h.pSaveIndexData := ADR(G_CANopen_CAN3.SaveData[0]);
G_CANopen_CAN3.SaveData[3].itfSaveAll := G_CANopen_CAN3.SaveAll;
G_CANopen_CAN3.SaveData[3].itfDeleteAll := G_CANopen_CAN3.DeleteAll;
G_CANopen_CAN3.OD.pAdditionalData := ADR(G_CANopen_CAN3.SaveSubData1010h);

IF G_CANopen_CAN3_VAR.OD_Error = EPEC_CANopen.Errors.NoError THEN
	G_CANopen_CAN3.Initialize(i_pOD:=ADR(G_CANopen_CAN3.OD), i_pParamHandler:=ADR(G_Common.ParHandler), o_Error => G_CANopen_CAN3_VAR.ODSave_Error);
END_IF

(* Check all protocol init status flags *)
IF G_CANopen_CAN3_VAR.NMT_Error = EPEC_CANopen.Errors.NoError AND
	G_CANopen_CAN3_VAR.SSDO_Error = EPEC_CANopen.Errors.NoError AND
	G_CANopen_CAN3_VAR.OD_Error = EPEC_CANopen.Errors.NoError AND
	G_CANopen_CAN3_VAR.HB_Error = EPEC_CANopen.Errors.NoError AND
	G_CANopen_CAN3_VAR.CSDO_Error = EPEC_CANopen.Errors.NoError AND
	G_CANopen_CAN3_VAR.GFC_Error = EPEC_CANopen.Errors.NoError
THEN
	G_InitCANopenCan3Error := FALSE; (* No errors in protocol inits *)
ELSE
	G_InitCANopenCan3Error := TRUE;
END_IF



G_InitProtocolsCan3State := InitCanProtocolStates.INIT_J1939;

InitCanProtocolStates.INIT_J1939:



                  
G_InitProtocolsCan3State := InitCanProtocolStates.INIT_PROTOCOLS_DONE;

InitCanProtocolStates.INIT_PROTOCOLS_DONE:
G_InitProtocolsCan3Ready:=TRUE;
END_CASE
END_ACTION

ACTION Init_Protocols_Can4_Action:
(*###########################################################*)
(*This block is created implicit. Don't add own code to here.*)
(*###########################################################*)
;
CASE G_InitProtocolsCan4State OF

InitCanProtocolStates.INIT_CANOPEN_PROTOCOLS:
(*CAN4 INIT*)

G_CANopen_CAN4.Device.itfCanChannel:=G_CAN4_Channel; (*Connect device to can channel*)
G_CANopen_CAN4.Device.NodeID := BYTE#1;
G_CANopen_CAN4.NMT.NmtState:=EPEC_CANopen.NMTState.BootUp; (* Set NMT status to BOOTUP *)

(*Initialize OD's data structures*)
G_CANopen_CAN4.OD.EntryCount:=SIZEOF(G_CANopen_CAN4.ODEntrys)/SIZEOF(G_CANopen_CAN4.ODEntrys[1]); (*Max entries of given OD(CANopenDeviceODEntrys array)*)
G_CANopen_CAN4.OD.InOrder:=FALSE; (*OD isn't in order*)
G_CANopen_CAN4.OD.NextFree:=0; (*OD does not have any entries yet*)
G_CANopen_CAN4.OD.pODEntry:=ADR(G_CANopen_CAN4.ODEntrys); (*Pointer to OD array*)

(*Define NMT protocol*)
G_CANopen_CAN4.Protocols[1].Protocol:=EPEC_CANopen.ProtocolType.NMT;
G_CANopen_CAN4.Protocols[1].pData:=ADR(G_CANopen_CAN4.NMT);
G_CANopen_CAN4.Protocols[1].itfProtocol:=G_CANopen_CAN4.NMT_Handler;
G_CANopen_CAN4.Protocols[1].pError:=ADR(G_CANopen_CAN4_VAR.NMT_Error);
G_CANopen_CAN4_VAR.ProtocolAdded[1] := CANopenDeviceAddProtocol( (* Add to protocol stack *)
	i_pDevice:=ADR(G_CANopen_CAN4.Device),
	i_pProtocol:=ADR(G_CANopen_CAN4.Protocols[1]),
);

(*Initialize NMT protocol*)
IF G_CANopen_CAN4_VAR.ProtocolAdded[1] THEN
	G_CANopen_CAN4.NMT_Handler.Init(
		i_pDevice := ADR(G_CANopen_CAN4.Device),
		i_ThisIsMaster := FALSE,
		i_StartInterval :=  1000,
		i_pMonitoredNodes := 0,
		i_NumberOfNodes := 0,
		i_SimultaneousSlaveConfiguration := FALSE,
		o_Error => G_CANopen_CAN4_VAR.NMT_Error
	);
ELSE
	G_CANopen_CAN4_VAR.NMT_Error := EPEC_CANopen.Errors.ProtocolDataMissing;
END_IF

(*Define OD protocol*)
G_CANopen_CAN4.Protocols[2].Protocol:=EPEC_CANopen.ProtocolType.OD;
G_CANopen_CAN4.Protocols[2].pData:=ADR(G_CANopen_CAN4.OD);
G_CANopen_CAN4.Protocols[2].pError:=ADR(G_CANopen_CAN4_VAR.OD_Error);
G_CANopen_CAN4_VAR.ProtocolAdded[2] := CANopenDeviceAddProtocol( (* Add to protocol stack *)
	i_pDevice:=ADR(G_CANopen_CAN4.Device),
	i_pProtocol:=ADR(G_CANopen_CAN4.Protocols[2]),
);
IF NOT G_CANopen_CAN4_VAR.ProtocolAdded[2] THEN
	G_CANopen_CAN4_VAR.OD_Error := EPEC_CANopen.Errors.ProtocolDataMissing;
END_IF

(*Define HB protocol
- Uses NMT and OD protocol data, thus need to be defined after them.
*)
G_CANopen_CAN4.HB.HeartBeat.PT := T#200MS; (* HB producer time *)

G_CANopen_CAN4.Protocols[3].Protocol:=EPEC_CANopen.ProtocolType.HB;
G_CANopen_CAN4.Protocols[3].pData:=ADR(G_CANopen_CAN4.HB);
G_CANopen_CAN4.Protocols[3].itfProtocol:=G_CANopen_CAN4.HB_Handler;
G_CANopen_CAN4.Protocols[3].pError:=ADR(G_CANopen_CAN4_VAR.HB_Error);
G_CANopen_CAN4_VAR.ProtocolAdded[3] := CANopenDeviceAddProtocol( (* Add to protocol stack *)
	i_pDevice:=ADR(G_CANopen_CAN4.Device),
	i_pProtocol:=ADR(G_CANopen_CAN4.Protocols[3]),
);

(* Initialize HB protocol *)
IF G_CANopen_CAN4_VAR.ProtocolAdded[3] THEN
	G_CANopen_CAN4.HB_Handler.Init(
		i_pDevice := ADR(G_CANopen_CAN4.Device),
		o_Error => G_CANopen_CAN4_VAR.HB_Error
	);

	(* Add monitored nodes *)
ELSE
	G_CANopen_CAN4_VAR.HB_Error := EPEC_CANopen.Errors.ProtocolDataMissing;
END_IF

(*Define SSDO protocol*)
G_CANopen_CAN4.Protocols[4].Protocol:=EPEC_CANopen.ProtocolType.SSDO;
G_CANopen_CAN4.Protocols[4].pData:=ADR(G_CANopen_CAN4.SSDO);
G_CANopen_CAN4.Protocols[4].itfProtocol:=G_CANopen_CAN4.SSDO_Handler;
G_CANopen_CAN4.Protocols[4].pError:=ADR(G_CANopen_CAN4_VAR.SSDO_Error);
G_CANopen_CAN4_VAR.ProtocolAdded[4] := CANopenDeviceAddProtocol( (* Add to protocol stack *)
	i_pDevice:=ADR(G_CANopen_CAN4.Device),
	i_pProtocol:=ADR(G_CANopen_CAN4.Protocols[4])
);
IF G_CANopen_CAN4_VAR.ProtocolAdded[4] THEN
	G_CANopen_CAN4.SSDO_Handler.Init(
		i_pDevice := ADR(G_CANopen_CAN4.Device),
		o_Error => G_CANopen_CAN4_VAR.SSDO_Error
	);
ELSE
	G_CANopen_CAN4_VAR.SSDO_Error := EPEC_CANopen.Errors.ProtocolDataMissing;
END_IF

(*Define GFC protocol*)
G_CANopen_CAN4.Protocols[5].Protocol:=EPEC_CANopen.ProtocolType.GFC;
G_CANopen_CAN4.Protocols[5].pData:=ADR(G_CANopen_CAN4.GFC);
G_CANopen_CAN4.Protocols[5].itfProtocol:=G_CANopen_CAN4.GFC_Handler;
G_CANopen_CAN4.Protocols[5].pError:=ADR(G_CANopen_CAN4_VAR.GFC_Error);
G_CANopen_CAN4_VAR.ProtocolAdded[5] := CANopenDeviceAddProtocol(  (* Add to protocol stack *)
	i_pDevice:=ADR(G_CANopen_CAN4.Device),
	i_pProtocol:=ADR(G_CANopen_CAN4.Protocols[5])
);
IF G_CANopen_CAN4_VAR.ProtocolAdded[5] THEN
	G_CANopen_CAN4.GFC_Handler.Init(
		i_pDevice := ADR(G_CANopen_CAN4.Device),
		i_pStatus:=ADR(G_CANopen_CAN4_VAR.GFC_Status),
		o_Error => G_CANopen_CAN4_VAR.GFC_Error
	);
ELSE
	G_CANopen_CAN4_VAR.GFC_Error := EPEC_CANopen.Errors.ProtocolDataMissing;
END_IF

(* Init CSDO instance array for bus *)
EPEC_CANopen.CANopenSDOManager.Init(
	i_pDevice:=ADR(G_CANopen_CAN4.Device),
	i_NodeId:=G_CANopen_CAN4.Device.NodeID,
	i_pCsdoArrayStart:=ADR(G_CANopen_CAN4.CSDOS),
	i_CsdoArraySize:=127,
	o_Error=>G_CANopen_CAN4_VAR.CSDO_Error
);





G_InitProtocolsCan4State := InitCanProtocolStates.INIT_CANOPEN_OD;

InitCanProtocolStates.INIT_CANOPEN_OD:

(*16#0001..16#0009 Default types *)
G_CANopen_CAN4_VAR.OD_Error := EPEC_CANopen.CANopenODAddDefautTypes(
	i_pOD:= ADR(G_CANopen_CAN4.OD)
);

(* 16#1000 Information about the device type *)
IF G_CANopen_CAN4_VAR.OD_Error = EPEC_CANopen.Errors.NoError THEN
	G_CANopen_CAN4_VAR.OD_Error := CANopenODAddLine(
		i_pOD := ADR(G_CANopen_CAN4.OD),(*Address of Object dictionary where index will be added*)
		i_Index := G_CANOPEN_ODINDEX_DEVICE_TYPE,
		i_ObjectCode := EPEC_CANopen.ObjectCode.OD_VAR,(*Type of index*)
		i_NumOfSubids := USINT#0,(*Number of subindexes*)
		i_TypeSpec := EPEC_CANopen.DataType.Deftype_UNSIGNED32,(*Index datatype, either user defined or standard CiA 301*)
		i_ObjectAccess := G_CANOPEN_OD_ACCESS_NOWRITE OR G_CANOPEN_OD_ACCESS_SUB0NOWRITE,
		i_Sub0data := USINT#0,(*Value of subindex0 in array or (def)struct*)
		i_pIndexData := ADR(G_CAN4_VAR.DeviceType_Device4),
		i_itfSDOHandler := DWORD#0
	);
END_IF

(* 16#1001 Error information *)
IF G_CANopen_CAN4_VAR.OD_Error = EPEC_CANopen.Errors.NoError THEN
	G_CANopen_CAN4_VAR.OD_Error := CANopenODAddLine(
		i_pOD := ADR(G_CANopen_CAN4.OD),(*Address of Object dictionary where index will be added*)
		i_Index := G_CANOPEN_ODINDEX_ERROR_REGISTER,
		i_ObjectCode := EPEC_CANopen.ObjectCode.OD_VAR,(*Type of index*)
		i_NumOfSubids := USINT#0,(*Number of subindexes*)
		i_TypeSpec := EPEC_CANopen.DataType.Deftype_UNSIGNED8,(*Index datatype, either user defined or standard CiA 301*)
		i_ObjectAccess := G_CANOPEN_OD_ACCESS_NOWRITE OR G_CANOPEN_OD_ACCESS_SUB0NOWRITE,
		i_Sub0data := USINT#0,(*Value of subindex0 in array or (def)struct*)
		i_pIndexData := ADR(G_CAN4_VAR.ErrorReg_Device4),
		i_itfSDOHandler := DWORD#0
	);
END_IF

(* 16#100A Manufacturer software version *)
IF G_CANopen_CAN4_VAR.OD_Error = EPEC_CANopen.Errors.NoError THEN
	G_CANopen_CAN4_VAR.OD_Error := CANopenODAddLine(
		i_pOD := ADR(G_CANopen_CAN4.OD),(*Address of Object dictionary where index will be added*)
		i_Index := G_CANOPEN_ODINDEX_MF_SW_VERSION,
		i_ObjectCode := EPEC_CANopen.ObjectCode.OD_VAR,(*Type of index*)
		i_NumOfSubids := USINT#0,(*Number of subindexes*)
		i_TypeSpec := EPEC_CANopen.DataType.Deftype_STRING,(*Index datatype, either user defined or standard CiA 301*)
		i_ObjectAccess := G_CANOPEN_OD_ACCESS_NOWRITE OR G_CANOPEN_OD_ACCESS_SUB0NOWRITE,
		i_Sub0data := USINT#0,(*Value of subindex0 in array or (def)struct*)
		i_pIndexData := ADR(G_SystemInfo.SWVersion),
		i_itfSDOHandler := DWORD#0
	);
END_IF

(* 16#1018   Vendor ID *)
IF G_CANopen_CAN4_VAR.OD_Error = EPEC_CANopen.Errors.NoError THEN
	G_CANopen_CAN4_VAR.OD_Error := CANopenODAddLine(
		i_pOD := ADR(G_CANopen_CAN4.OD),(*Address of Object dictionary where index will be added*)
		i_index := G_CANOPEN_ODINDEX_IDENTITY_OBJECT,
		i_ObjectCode := EPEC_CANopen.ObjectCode.OD_ARRAY, (*Type of index*)
		i_NumOfSubids := USINT#4,(*Number of subindexes*)
		i_TypeSpec := EPEC_CANopen.DataType.Deftype_UNSIGNED32,(*Index of 16-bit deftype*)
		i_ObjectAccess := G_CANOPEN_OD_ACCESS_NOWRITE OR G_CANOPEN_OD_ACCESS_SUB0NOWRITE,
		i_sub0data := USINT#4,(*Value of subindex0 in array or (def)struct*)
		i_pIndexData := ADR(G_SystemInfo.Identity),
		i_itfSDOHandler := DWORD#0
	);
END_IF
(* 16#2129 PDO Dummy Variable Index *)
IF G_CANopen_CAN4_VAR.OD_Error = EPEC_CANopen.Errors.NoError THEN
	G_CANopen_CAN4_VAR.OD_Error := CANopenODAddLine(
		i_pOD := ADR(G_CANopen_CAN4.OD),(*Address of Object dictionary where index will be added*)
		i_Index := 16#2129,
		i_ObjectCode := EPEC_CANopen.ObjectCode.OD_VAR,(*Type of index*)
		i_NumOfSubids := USINT#0,(*Number of subindexes*)
		i_TypeSpec := EPEC_CANopen.DataType.Deftype_UNSIGNED8,(*Index datatype, either user defined or standard CiA 301*)
		i_ObjectAccess := G_CANOPEN_OD_ACCESS_READWRITE,
		i_Sub0data := USINT#0,(*Value of subindex0 in array or (def)struct*)
		i_pIndexData := ADR(G_CAN4_VAR.CAN4_PDO_DUMMY),
		i_itfSDOHandler := DWORD#0
	);
END_IF

(* 16#2130   Application version *)
IF G_CANopen_CAN4_VAR.OD_Error = EPEC_CANopen.Errors.NoError THEN
	G_CANopen_CAN4_VAR.OD_Error := CANopenODAddLine(
		i_pOD := ADR(G_CANopen_CAN4.OD),(*Address of Object dictionary where index will be added*)
		i_index := 16#2130,
		i_ObjectCode := EPEC_CANopen.ObjectCode.OD_ARRAY, (*Type of index*)
		i_NumOfSubids := USINT#10,(*Number of subindexes*)
		i_TypeSpec := EPEC_CANopen.DataType.Deftype_STRING,(*Index of 16-bit deftype*)
		i_ObjectAccess := G_CANOPEN_OD_ACCESS_NOWRITE OR G_CANOPEN_OD_ACCESS_SUB0NOWRITE,
		i_sub0data := USINT#10,(*Value of subindex0 in array or (def)struct*)
		i_pIndexData := ADR(G_SystemInfo.SoftwareInformation),
		i_itfSDOHandler := DWORD#0
	);
END_IF

(* 16#2131 Parameter CSV unique ID *)
IF G_CANopen_CAN4_VAR.OD_Error = EPEC_CANopen.Errors.NoError THEN
	G_CANopen_CAN4_VAR.OD_Error := CANopenODAddLine(
		i_pOD := ADR(G_CANopen_CAN4.OD),(*Address of Object dictionary where index will be added*)
		i_Index := 16#2131,
		i_ObjectCode := EPEC_CANopen.ObjectCode.OD_VAR,(*Type of index*)
		i_NumOfSubids := USINT#0,(*Number of subindexes*)
		i_TypeSpec := EPEC_CANopen.DataType.Deftype_UNSIGNED16,(*Index datatype, either user defined or standard CiA 301*)
		i_ObjectAccess := G_CANOPEN_OD_ACCESS_NOWRITE OR G_CANOPEN_OD_ACCESS_SUB0NOWRITE,
		i_Sub0data := USINT#0,(*Value of subindex0 in array or (def)struct*)
		i_pIndexData := ADR(G_CAN4_VAR.Parameter_CSV_unique_ID4),
		i_itfSDOHandler := DWORD#0
	);
END_IF



G_InitProtocolsCan4State := InitCanProtocolStates.INIT_CANOPEN_PDO;

InitCanProtocolStates.INIT_CANOPEN_PDO:



G_InitProtocolsCan4State := InitCanProtocolStates.INIT_CANOPEN_OD_SAVE;

InitCanProtocolStates.INIT_CANOPEN_OD_SAVE:

(*Initialize OD save*)
G_CANopen_CAN4.SaveAll.Init(i_pParamHandler:=ADR(G_Common.ParHandler));
G_CANopen_CAN4.DeleteAll.Init(i_pParamHandler:=ADR(G_Common.ParHandler));
G_CANopen_CAN4.SaveSubData1010h.pSaveSigns := ADR(G_CANopen_CAN4_VAR.SaveSigns1010[0]);
G_CANopen_CAN4.SaveSubData1010h.NumOfEntrys := 4;
G_CANopen_CAN4.SaveSubData1010h.pSaveIndexData := ADR(G_CANopen_CAN4.SaveData[0]);
G_CANopen_CAN4.SaveData[3].itfSaveAll := G_CANopen_CAN4.SaveAll;
G_CANopen_CAN4.SaveData[3].itfDeleteAll := G_CANopen_CAN4.DeleteAll;
G_CANopen_CAN4.OD.pAdditionalData := ADR(G_CANopen_CAN4.SaveSubData1010h);

IF G_CANopen_CAN4_VAR.OD_Error = EPEC_CANopen.Errors.NoError THEN
	G_CANopen_CAN4.Initialize(i_pOD:=ADR(G_CANopen_CAN4.OD), i_pParamHandler:=ADR(G_Common.ParHandler), o_Error => G_CANopen_CAN4_VAR.ODSave_Error);
END_IF

(* Check all protocol init status flags *)
IF G_CANopen_CAN4_VAR.NMT_Error = EPEC_CANopen.Errors.NoError AND
	G_CANopen_CAN4_VAR.SSDO_Error = EPEC_CANopen.Errors.NoError AND
	G_CANopen_CAN4_VAR.OD_Error = EPEC_CANopen.Errors.NoError AND
	G_CANopen_CAN4_VAR.HB_Error = EPEC_CANopen.Errors.NoError AND
	G_CANopen_CAN4_VAR.CSDO_Error = EPEC_CANopen.Errors.NoError AND
	G_CANopen_CAN4_VAR.GFC_Error = EPEC_CANopen.Errors.NoError
THEN
	G_InitCANopenCan4Error := FALSE; (* No errors in protocol inits *)
ELSE
	G_InitCANopenCan4Error := TRUE;
END_IF



G_InitProtocolsCan4State := InitCanProtocolStates.INIT_J1939;

InitCanProtocolStates.INIT_J1939:

(* EBC1 *)
J1939_CAN4.In.ABS1.PGN_EBC1.pSPNs:=ADR(J1939_CAN4.In.ABS1.PGN_EBC1_SPNs);
J1939_CAN4.In.ABS1.PGN_EBC1.PGN_Number:=16#F001;
J1939_CAN4.In.ABS1.PGN_EBC1.SourceAddress:=16#000B;
J1939_CAN4.In.ABS1.PGN_EBC1.Destination:=16#00FF;
J1939_CAN4.In.ABS1.PGN_EBC1.CycleTime:=100;
J1939_CAN4.In.ABS1.PGN_EBC1.DataPage:=0;
J1939_CAN4.In.ABS1.PGN_EBC1.NumberOfSPNs:=23;
J1939_CAN4.In.ABS1.PGN_EBC1.Priority:=6;
J1939_CAN4.In.ABS1.PGN_EBC1.DataLength:=8;

	J1939_CAN4.In.ABS1.PGN_EBC1_SPNs[1].Size:=2; (* BYTE *)
	J1939_CAN4.In.ABS1.PGN_EBC1_SPNs[1].pData:=ADR(J1939_CAN4.In.ABS1.EBC1_ASREngCtrlActive);
	J1939_CAN4.In.ABS1.PGN_EBC1_SPNs[2].Size:=2; (* BYTE *)
	J1939_CAN4.In.ABS1.PGN_EBC1_SPNs[2].pData:=ADR(J1939_CAN4.In.ABS1.EBC1_ASRBrakeCtrlActive);
	J1939_CAN4.In.ABS1.PGN_EBC1_SPNs[3].Size:=2; (* BYTE *)
	J1939_CAN4.In.ABS1.PGN_EBC1_SPNs[3].pData:=ADR(J1939_CAN4.In.ABS1.EBC1_AntiLockBrakingActive);
	J1939_CAN4.In.ABS1.PGN_EBC1_SPNs[4].Size:=2; (* BYTE *)
	J1939_CAN4.In.ABS1.PGN_EBC1_SPNs[4].pData:=ADR(J1939_CAN4.In.ABS1.EBC1_EBSBrakeSwitch);
	J1939_CAN4.In.ABS1.PGN_EBC1_SPNs[5].Size:=8; (* BYTE *)
	J1939_CAN4.In.ABS1.PGN_EBC1_SPNs[5].pData:=ADR(J1939_CAN4.In.ABS1.EBC1_BrakePedalPos);
	J1939_CAN4.In.ABS1.PGN_EBC1_SPNs[6].Size:=2; (* BYTE *)
	J1939_CAN4.In.ABS1.PGN_EBC1_SPNs[6].pData:=ADR(J1939_CAN4.In.ABS1.EBC1_ABSOffroadSwitch);
	J1939_CAN4.In.ABS1.PGN_EBC1_SPNs[7].Size:=2; (* BYTE *)
	J1939_CAN4.In.ABS1.PGN_EBC1_SPNs[7].pData:=ADR(J1939_CAN4.In.ABS1.EBC1_ASROffroadSwitch);
	J1939_CAN4.In.ABS1.PGN_EBC1_SPNs[8].Size:=2; (* BYTE *)
	J1939_CAN4.In.ABS1.PGN_EBC1_SPNs[8].pData:=ADR(J1939_CAN4.In.ABS1.EBC1_ASRHillHolderSwitch);
	J1939_CAN4.In.ABS1.PGN_EBC1_SPNs[9].Size:=2; (* BYTE *)
	J1939_CAN4.In.ABS1.PGN_EBC1_SPNs[9].pData:=ADR(J1939_CAN4.In.ABS1.EBC1_TractionCtrlOverrideSwitch);
	J1939_CAN4.In.ABS1.PGN_EBC1_SPNs[10].Size:=2; (* BYTE *)
	J1939_CAN4.In.ABS1.PGN_EBC1_SPNs[10].pData:=ADR(J1939_CAN4.In.ABS1.EBC1_AccelInterlockSwitch);
	J1939_CAN4.In.ABS1.PGN_EBC1_SPNs[11].Size:=2; (* BYTE *)
	J1939_CAN4.In.ABS1.PGN_EBC1_SPNs[11].pData:=ADR(J1939_CAN4.In.ABS1.EBC1_EngDerateSwitch);
	J1939_CAN4.In.ABS1.PGN_EBC1_SPNs[12].Size:=2; (* BYTE *)
	J1939_CAN4.In.ABS1.PGN_EBC1_SPNs[12].pData:=ADR(J1939_CAN4.In.ABS1.EBC1_EngAuxEngShutdownSwitch);
	J1939_CAN4.In.ABS1.PGN_EBC1_SPNs[13].Size:=2; (* BYTE *)
	J1939_CAN4.In.ABS1.PGN_EBC1_SPNs[13].pData:=ADR(J1939_CAN4.In.ABS1.EBC1_RemoteAccelEnableSwitch);
	J1939_CAN4.In.ABS1.PGN_EBC1_SPNs[14].Size:=8; (* BYTE *)
	J1939_CAN4.In.ABS1.PGN_EBC1_SPNs[14].pData:=ADR(J1939_CAN4.In.ABS1.EBC1_EngRetarderSelection);
	J1939_CAN4.In.ABS1.PGN_EBC1_SPNs[15].Size:=2; (* BYTE *)
	J1939_CAN4.In.ABS1.PGN_EBC1_SPNs[15].pData:=ADR(J1939_CAN4.In.ABS1.EBC1_ABSFullyOperational);
	J1939_CAN4.In.ABS1.PGN_EBC1_SPNs[16].Size:=2; (* BYTE *)
	J1939_CAN4.In.ABS1.PGN_EBC1_SPNs[16].pData:=ADR(J1939_CAN4.In.ABS1.EBC1_EBSRedWarningSignal);
	J1939_CAN4.In.ABS1.PGN_EBC1_SPNs[17].Size:=2; (* BYTE *)
	J1939_CAN4.In.ABS1.PGN_EBC1_SPNs[17].pData:=ADR(J1939_CAN4.In.ABS1.EBC1_ABS_EBSAmberWarningSignal);
	J1939_CAN4.In.ABS1.PGN_EBC1_SPNs[18].Size:=2; (* BYTE *)
	J1939_CAN4.In.ABS1.PGN_EBC1_SPNs[18].pData:=ADR(J1939_CAN4.In.ABS1.EBC1_ATC_ASRInformationSignal);
	J1939_CAN4.In.ABS1.PGN_EBC1_SPNs[19].Size:=8; (* BYTE *)
	J1939_CAN4.In.ABS1.PGN_EBC1_SPNs[19].pData:=ADR(J1939_CAN4.In.ABS1.EBC1_SrcAddrssOfCtrllngDvcFrBrkCntrl);
	J1939_CAN4.In.ABS1.PGN_EBC1_SPNs[20].Size:=2; (* BYTE *)
	J1939_CAN4.In.ABS1.PGN_EBC1_SPNs[20].pData:=ADR(J1939_CAN4.In.ABS1.J1939_CAN4_EBC1_Dummy_RX_1);
	J1939_CAN4.In.ABS1.PGN_EBC1_SPNs[21].Size:=2; (* BYTE *)
	J1939_CAN4.In.ABS1.PGN_EBC1_SPNs[21].pData:=ADR(J1939_CAN4.In.ABS1.EBC1_HaltBrakeSwitch);
	J1939_CAN4.In.ABS1.PGN_EBC1_SPNs[22].Size:=2; (* BYTE *)
	J1939_CAN4.In.ABS1.PGN_EBC1_SPNs[22].pData:=ADR(J1939_CAN4.In.ABS1.EBC1_TrailerABSStatus);
	J1939_CAN4.In.ABS1.PGN_EBC1_SPNs[23].Size:=2; (* BYTE *)
	J1939_CAN4.In.ABS1.PGN_EBC1_SPNs[23].pData:=ADR(J1939_CAN4.In.ABS1.EBC1_TrctrMntdTrilerABSWarningSignal);
(* TD *)
J1939_CAN4.In.Tacho.PGN_TD.pSPNs:=ADR(J1939_CAN4.In.Tacho.PGN_TD_SPNs);
J1939_CAN4.In.Tacho.PGN_TD.PGN_Number:=16#FEE6;
J1939_CAN4.In.Tacho.PGN_TD.SourceAddress:=16#00EE;
J1939_CAN4.In.Tacho.PGN_TD.Destination:=16#00FF;
J1939_CAN4.In.Tacho.PGN_TD.CycleTime:=0;
J1939_CAN4.In.Tacho.PGN_TD.DataPage:=0;
J1939_CAN4.In.Tacho.PGN_TD.NumberOfSPNs:=8;
J1939_CAN4.In.Tacho.PGN_TD.Priority:=6;
J1939_CAN4.In.Tacho.PGN_TD.DataLength:=8;

	J1939_CAN4.In.Tacho.PGN_TD_SPNs[1].Size:=8; (* BYTE *)
	J1939_CAN4.In.Tacho.PGN_TD_SPNs[1].pData:=ADR(J1939_CAN4.In.Tacho.TD_Seconds);
	J1939_CAN4.In.Tacho.PGN_TD_SPNs[2].Size:=8; (* BYTE *)
	J1939_CAN4.In.Tacho.PGN_TD_SPNs[2].pData:=ADR(J1939_CAN4.In.Tacho.TD_Minutes);
	J1939_CAN4.In.Tacho.PGN_TD_SPNs[3].Size:=8; (* BYTE *)
	J1939_CAN4.In.Tacho.PGN_TD_SPNs[3].pData:=ADR(J1939_CAN4.In.Tacho.TD_Hours);
	J1939_CAN4.In.Tacho.PGN_TD_SPNs[4].Size:=8; (* BYTE *)
	J1939_CAN4.In.Tacho.PGN_TD_SPNs[4].pData:=ADR(J1939_CAN4.In.Tacho.TD_Month);
	J1939_CAN4.In.Tacho.PGN_TD_SPNs[5].Size:=8; (* BYTE *)
	J1939_CAN4.In.Tacho.PGN_TD_SPNs[5].pData:=ADR(J1939_CAN4.In.Tacho.TD_Day);
	J1939_CAN4.In.Tacho.PGN_TD_SPNs[6].Size:=8; (* BYTE *)
	J1939_CAN4.In.Tacho.PGN_TD_SPNs[6].pData:=ADR(J1939_CAN4.In.Tacho.TD_Year);
	J1939_CAN4.In.Tacho.PGN_TD_SPNs[7].Size:=8; (* BYTE *)
	J1939_CAN4.In.Tacho.PGN_TD_SPNs[7].pData:=ADR(J1939_CAN4.In.Tacho.TD_LocalMinuteOffset);
	J1939_CAN4.In.Tacho.PGN_TD_SPNs[8].Size:=8; (* BYTE *)
	J1939_CAN4.In.Tacho.PGN_TD_SPNs[8].pData:=ADR(J1939_CAN4.In.Tacho.TD_LocalHourOffset);
(* VD *)
J1939_CAN4.In.Tacho.PGN_VD.pSPNs:=ADR(J1939_CAN4.In.Tacho.PGN_VD_SPNs);
J1939_CAN4.In.Tacho.PGN_VD.PGN_Number:=16#FEE0;
J1939_CAN4.In.Tacho.PGN_VD.SourceAddress:=16#00EE;
J1939_CAN4.In.Tacho.PGN_VD.Destination:=16#00FF;
J1939_CAN4.In.Tacho.PGN_VD.CycleTime:=100;
J1939_CAN4.In.Tacho.PGN_VD.DataPage:=0;
J1939_CAN4.In.Tacho.PGN_VD.NumberOfSPNs:=2;
J1939_CAN4.In.Tacho.PGN_VD.Priority:=6;
J1939_CAN4.In.Tacho.PGN_VD.DataLength:=8;

	J1939_CAN4.In.Tacho.PGN_VD_SPNs[1].Size:=32; (* DWORD *)
	J1939_CAN4.In.Tacho.PGN_VD_SPNs[1].pData:=ADR(J1939_CAN4.In.Tacho.VD_TripDistance);
	J1939_CAN4.In.Tacho.PGN_VD_SPNs[2].Size:=32; (* DWORD *)
	J1939_CAN4.In.Tacho.PGN_VD_SPNs[2].pData:=ADR(J1939_CAN4.In.Tacho.VD_TotalVehicleDistance);

J1939_CAN4.In.PGNs[1].pPGN:=ADR(J1939_CAN4.In.ABS1.PGN_EBC1);
J1939_CAN4.In.PGNs[2].pPGN:=ADR(J1939_CAN4.In.Tacho.PGN_TD);
J1939_CAN4.In.PGNs[3].pPGN:=ADR(J1939_CAN4.In.Tacho.PGN_VD);

                  
G_InitProtocolsCan4State := InitCanProtocolStates.INIT_PROTOCOLS_DONE;

InitCanProtocolStates.INIT_PROTOCOLS_DONE:
G_InitProtocolsCan4Ready:=TRUE;
END_CASE
END_ACTION

